FUNCTION_BLOCK "GCS7_GrpCtrlMain"	// FB 9
TITLE = Group Control UL
//
//COPYRIGHT:   (C) 1997 BY  BUHLER LTD
//                          CH-9240 UZWIL  SWITZERLAND
//
//PRODUCT:     GCS90
//
//TITLE:       FB 009 METHODS  OF  GROUPMANAGEMENT  with 320 groups
//                    Methoden der Gruppenverwaltung
//                    GCPROVB Revision =2
//-------------------------------------------------------------------------
//
//IDENT:        AUTOR:              DEPT:                           DATE:
//
//FB009.4.3     A.Egli              CT3                             23-Nov-2004
//              OutAutostartOkAll
//FB009.4.2     A.Egli              CT3                             14-Mar-2004
//              Reset Idling when group is externel used 
//FB009.4.1     A.Egli              CT3                             04-Mar-2004
//              Autostart: Filter with not ParNotRelForFault and 
//                                         ParNotRelForStarted
//FB009.4.0     A.Egli              CT3                             11-Nov-2003
//              OutAutoStartOkShared
//FB009.3.6     A.Egli              CT3                             14-Okt-2003
//              For available test use InExternal and not InLocked 
//FB009.3.5     A.Egli              CT3                             21-Aug-2003
//              Command OutAnyFault 
//FB009.3.4     A.Egli              CT3                             11-Aug-2003
//              Command CmdManualOffRel: 
//              Send command only to selected group, which OutShared=false
//FB009.3.3     A.Egli              CT3                             22-Jul-2003
//              Condition for All.OutStartWarning 
//FB009.3.2     A.Egli              CT3                             19-Mai-2003
//              OutStartwarning 
//FB009.3.1     A.Egli              CT3                             25-Mar-2003
//              OutPreStarted 
//FB009.3.0     A.Egli              CT3                             23-Sept-2002
//              New Relesae: 
//              OutLoaded;OutDPFault;OutHWStop;OutAutoStartOk; 
//              CmdContinue;InPreStart
//FB009.2.0     A.Egli              CT3                             13-Sept-2000
//              -320 group
//              -Any offset in section DB  
//              -Methode Code=0: Set Pointer 
//FB009.1.7     A.Egli              CT3                             13-Sept-2000
//              OutShared: Wrong pointer (DID with D replaced)
//FB009.1.6     A.Egli              CT3                             06-Jan-99
//              Warning if group with not rel. for fault is in state StFault
//FB009.1.5     A.Egli              CT3                             05-Jan-99
//              Warning if group with not rel. for fault is in state StFault
//FB009.1D      A.Egli              CT3                             20-Aug-99
//              OutFaultAll,FaultReset 
//FB009.1C      A.Egli              CT3                             18-Jul-99
//              OutWarning: Label wrong
//FB009.1B      A.Egli              CT3                             14-Okt-98
//              Reset InPreselected
//FB009.1A      A.Egli              AEE61                           13-Jun-96
//              1st Release
//
//-------------------------------------------------------------------------
//
//PURPOSE:            MANUAL : ....... .DOC
//                    CODE   : FB ...
//
//RESTRICTIONS: GCPROVB Revision >=2
//            
//-------------------------------------------------------------------------
//
//Calling convention:
//==================
//
//Actual open DB = Section DB
//
//Input parameter:
//===============
//CODE:
//  0 - Methode Set Pointer
//  1 - Methode InitPreselection
//  2 - Methode Selection
//  3 - Methode Deselection
//  4 - Methode UpdateCmdSt
//  5 - Methode UpdateEnable
//  6 - Methode UpdateOccupied
//
//Calling order for select of new groups:
//---------------------------------------
//1. Call Methode InitPreselection
//2. ASW: Prepare patter Sec.Gr.InPreselect 
//3. Call Methode Selection
//   ReturnValue: All.OutGrConflict
//4. Call ASW routine 'Select'
//
AUTHOR : EA
FAMILY : GCS7UL
NAME : GRVWMAIN
VERSION : 4.3
VAR_INPUT
  Code : INT ;	//0=Init,1=InitPreselect,2=Select,3=Deselect,4=UpdateCmdSt,5=UpdateEnable
END_VAR
VAR_IN_OUT
  Sec : UDT 20090;
END_VAR
VAR
  Spare : WORD ;
  All : STRUCT
   CmdClearIdling : BOOL ;	//Stop al groups of this section which are in idling
   OutAutoStartOkShared : BOOL ;
   InASWFlagAutostart : BOOL ;	//Free for ASW
   OutAutostartOkAll : BOOL ;	//Autostart of all selected groups ok
   Spare04 : BOOL ;
   Spare05 : BOOL ;
   OutPreStarted : BOOL ;
   OutPreStarting : BOOL ;	//Any group is pre-starting
   Spare10 : BOOL ;
   CmdContinue : BOOL ;	//(*new*)
   CmdManualOffRel : BOOL ;	//(*new*)
   CmdFaultReset : BOOL ;	//Command to fault reset
   CmdManualOff : BOOL ;	//Switch off maunual mode of all object
   OutStartwarning : BOOL ;	//Any selected group is in startwarning mode
   OutManualAny : BOOL ;	//Any object of this PLC is in manual mode
   InOutASWSelectionOK : BOOL ;	//Used by ASW
   OutSelectionValid : BOOL ;	//Any object is occupied for this section
   CmdNewSelection : BOOL ;	//An new object is occupied
   OutGrConflict : BOOL ;	//An object is not available
   OutGrIsLocked : BOOL ;	//An object is locked by ASW
   OutAutoStartOk : BOOL ;	//(*new*) All relevant Groups are in mode AutoStart
   OutManual : BOOL ;	//Any object of this section is in manual mode
   OutDPFault : BOOL ;	//(*new*)
   OutHWStop : BOOL ;	//(*new*)
   OutStoppedRel : BOOL ;
   OutStoppedAll : BOOL ;
   OutLoaded : BOOL ;	//(*new*)
   OutFaultIdling : BOOL ;
   OutFaultRel : BOOL ;
   OutFaultAll : BOOL ;
   OutIdling : BOOL ;
   OutWarning : BOOL ;
  END_STRUCT ;
  Feed : STRUCT
   InEnable : BOOL ;
   Spare01 : BOOL ;
   CmdNext : BOOL ;
   Spare03 : BOOL ;
   Spare04 : BOOL ;
   Spare05 : BOOL ;
   Spare06 : BOOL ;
   Spare07 : BOOL ;
   OutStoppedRel : BOOL ;
   OutStoppedAll : BOOL ;
   OutStartedRel : BOOL ;
   OutFaultIdling : BOOL ;
   OutFaultRel : BOOL ;
   OutFaultAll : BOOL ;
   OutIdling : BOOL ;
   OutSelected : BOOL ;
  END_STRUCT ;
  Mgr : STRUCT
   InEnable : BOOL ;
   Spare01 : BOOL ;
   CmdNext : BOOL ;
   Spare03 : BOOL ;
   Spare04 : BOOL ;
   Spare05 : BOOL ;
   Spare06 : BOOL ;
   Spare07 : BOOL ;
   OutStoppedRel : BOOL ;
   OutStoppedAll : BOOL ;
   OutStartedRel : BOOL ;
   OutFaultIdling : BOOL ;
   OutFaultRel : BOOL ;
   OutFaultAll : BOOL ;
   OutIdling : BOOL ;
   OutSelected : BOOL ;
  END_STRUCT ;
  Wgr : STRUCT
   InEnable : BOOL ;
   Spare01 : BOOL ;
   CmdNext : BOOL ;
   Spare03 : BOOL ;
   Spare04 : BOOL ;
   Spare05 : BOOL ;
   Spare06 : BOOL ;
   Spare07 : BOOL ;
   OutStoppedRel : BOOL ;
   OutStoppedAll : BOOL ;
   OutStartedRel : BOOL ;
   OutFaultIdling : BOOL ;
   OutFaultRel : BOOL ;
   OutFaultAll : BOOL ;
   OutIdling : BOOL ;
   OutSelected : BOOL ;
  END_STRUCT ;
  Ggr : STRUCT
   InEnable : BOOL ;
   Spare01 : BOOL ;
   CmdNext : BOOL ;
   Spare03 : BOOL ;
   Spare04 : BOOL ;
   Spare05 : BOOL ;
   Spare06 : BOOL ;
   Spare07 : BOOL ;
   OutStoppedRel : BOOL ;
   OutStoppedAll : BOOL ;
   OutStartedRel : BOOL ;
   OutFaultIdling : BOOL ;
   OutFaultRel : BOOL ;
   OutFaultAll : BOOL ;
   OutIdling : BOOL ;
   OutSelected : BOOL ;
  END_STRUCT ;
  InPreselect : ARRAY  [1 .. 320 ] OF BOOL ;
  OutSelected : ARRAY  [1 .. 320 ] OF BOOL ;
  OutIdling : ARRAY  [1 .. 320 ] OF BOOL ;
  ParNotRelForStarted : ARRAY  [1 .. 320 ] OF BOOL  := TRUE;
  ParNotRelForFault : ARRAY  [1 .. 320 ] OF BOOL  := TRUE;
  InManual : ARRAY  [1 .. 320 ] OF BOOL  := FALSE;
  InPreStart : ARRAY  [1 .. 320 ] OF //Input from section: These groups are pre-starting
  BOOL  := FALSE;
END_VAR
VAR_TEMP
  TmpInOut : STRUCT 	//Methode 4:Temporare copy of input an output of the actual type
   InEnable : BOOL ;
   Spare01 : BOOL ;
   CmdNext : BOOL ;
   Spare03 : BOOL ;
   Spare04 : BOOL ;
   InManual : BOOL ;
   Spare06 : BOOL ;
   Spare07 : BOOL ;
   OutStoppedRel : BOOL ;
   OutStoppedAll : BOOL ;
   OutStartedRel : BOOL ;
   OutFaultIdling : BOOL ;
   OutFaultRel : BOOL ;
   OutFaultAll : BOOL ;
   OutIdling : BOOL ;
   OutSelected : BOOL ;
  END_STRUCT ;
  tmpAddrInOut : DINT ;	//Methode 4: Address of TmpInOut
  VarSelGrActType : DWORD ;	//Methode 4: Temporare pattern
  VarSelGrActTypeId : DWORD ;	//Methode 4: Temporare pattern Selected +idling
  tmpValue : DINT ;
  tmpCntLoopGr : BYTE ;
  tmpCntLoopType : BYTE ;
  tmpAddrLoop : DWORD ;
  tmpAddrSecPreselect : DWORD ;
  tmpAddrSecSelected : DWORD ;
  tmpAddrSecIdling : DWORD ;
  tmpAddrSecManual : DWORD ;
  tmpAddrSecParRelStarted : DWORD ;
  tmpAddrSecParRelFault : DWORD ;
  tmpAddrDB9ParXxx : DWORD ;	//Pointer parameter of group of type xxxx
  tmpAddrDB9ParXxxLoop : DWORD ;
  tmpAddrSecInPreStart : DWORD ;
  tmpCODE : INT ;	//FUNC
  SecArray : DINT ;	//Pointer to Array DB9.Section
  SecDB : INT ;	//Actual section DB
  tmpOffsetDI : DINT ;	//Offset Instanz
  tmpCodeIs5 : BOOL ;	//Methode Update Enable
  tmpSecByteNr : DINT ;
  tmpStoreAR2 : DWORD ;
  tmpInstanzDB : INT ;
  tmpNotRelevant : DWORD ;
  tmpNotRelevantForFault : DWORD ;
END_VAR
BEGIN
NETWORK
TITLE = Init Part 1
      L     #Code;
      T     #tmpCODE;
      L     P##Sec;
      LAR1;
//--- Section DB of actual instanz ----------
      L     W [AR1,P#0.0];
      T     #SecDB;
//--- Set Pointer to instanz in section DB ----------
      L     D [AR1,P#2.0];
      SLD   8;
      SRD   11;
      T     #tmpSecByteNr;
//------------------------------
      L     #tmpCODE;
      L     5;	// do not init for methode "Update Enable"
      ==I;
      =     #tmpCodeIs5;
      JC    InEn;
//--- Call Section DB ----------
      OPN   DI [#SecDB];
      L     #tmpSecByteNr;
      SLD   3;
      L     P##Code;
      +D;
      L     P##All;	//) Section DB has only UDT20090
      SLD   8;	//) Correction AR2 (10 Byte)
      SRD   8;	//)
      -D;	//)
      LAR2;	//-->Instanz
InEn: TAR2  #tmpStoreAR2;
NETWORK
TITLE = Methode "Set Pointer"
//=======================================================================
      OPN   "GCS7_GrCtrlDB";
      L     #tmpCODE;
      L     0;
      <>I;
      JC    iEnd;
//==========================================================
//Check DB9.ParMaxGroupCnt    : must be between 1 and 10
      L     10;
      L     "GCS7_GrCtrlDB".ParMaxGroupCnt;
      <I;
      JC    Stop;
      L     1;
      <I;
      JC    Stop;
//=======================================================================
//Enter ByteNumber in DB9.Section[x].DBB [<--2.0
      L     "GCS7_GrCtrlDB".ParByteNoSecDB;	// ) ParByteArraySectionDB
      SLD   3;
      LAR1;
iSLo: L     W#16#FFFF;	// )=  Sektion-List
      L     DBW [AR1,P#0.0];	// )
      ==I;
      JC    iAdd;	//-->Add pointer, if pointer is not found
      L     DINO;	//-->Actual Section-DB
      ==I;
      JC    iSOt;	//-->Enter pointer
      +AR1  P#4.0;
      JU    iSLo;
//=======================================================================
//"Add DB-Pointer"
iAdd: L     #SecDB;	//Bit-Number Section Interface
      T     DBW [AR1,P#0.0];	//DB9.Section[n].DBB
      L     W#16#FFFF;
      T     DBW [AR1,P#4.0];	//DB9.Section[n+1].DBB
//=======================================================================
//"Set Pointer"
iSOt: L     #tmpSecByteNr;	//Bit-Number Section Interface
      T     DBW [AR1,P#2.0];	//DB9.Section[x].DBB
      BEU;
//=======================================================================
//!!!!Call Stop, if DB is not found or AR2 < P#DIX2.0   !!!!!!!
//Note: 1. Check DB9.Section[x].DBB    : must be >1
//      2. Check DB9.ParMaxGroupCnt    : must be between 1 and 10
Stop: CALL  "SIEMENS_STP";
//=======================================================================
iEnd: NOP   0;
NETWORK
TITLE = Code=1: Methode "InitPreselection"
      L     #tmpCODE;	// )
      L     1;	// )
      <>I;	// )
      JC    aEnd;	// )
//-----------------------------------
//Init InPreselect
//Init InPreStart
      LAR1  AR2;
      L     P##InPreselect;
      +AR1;
      L     "GCS7_GrCtrlDB".ParMaxGroupCnt;
F1LE: T     #tmpCntLoopGr;
// Reset enable bit of selected groups
      L     0;
      T     DID [AR1,P#0.0];	//  )-> InPreselect
      T     DID [AR1,P#240.0];	//  )-> InPreStart (P#262.0- P#22.0 =+240.0)
      +AR1  P#4.0;
      L     #tmpCntLoopGr;
      LOOP  F1LE;
      JU    BACK;
aEnd: NOP   0;
NETWORK
TITLE =  FUNC=2: meth. "selection"
      L     #tmpCODE;
      L     2;
      <>I;
      JC    F2En;
//--- Available test--------   
      R     #All.OutGrConflict;
      R     #All.OutGrIsLocked;
      R     #All.CmdNewSelection;
      R     #All.OutPreStarting;
      OPN   "GCS7_GrCtrlDB";
      LAR1  P#0.0;	// Pointer to DB9
//=======================================================================
// 1. Test New Selection: 
// ---------------------
// 1.0 Set OutPreStarting
// 1.1 Set idling 
// 1.2 Test available
// 1.3 Deleselect Conficted groups 
// 1.4 Deselect not used groups
//=======================================================================
//==Begin Loop Goups A                  ===
      L     "GCS7_GrCtrlDB".ParMaxGroupCnt;
F2L1: T     #tmpCntLoopGr;
//--Pointer section
      TAR1;
      TAR2;
      +D;
      T     #tmpOffsetDI;
      L     P##InPreselect;
      +D;
      T     #tmpAddrSecPreselect;
// 
      L     #tmpOffsetDI;
      L     P##OutSelected;
      +D;
      T     #tmpAddrSecSelected;
// 
      L     #tmpOffsetDI;
      L     P##OutIdling;
      +D;
      T     #tmpAddrSecIdling;
// 
      L     #tmpOffsetDI;
      L     P##InPreStart;
      +D;
      T     #tmpAddrSecInPreStart;
// 
// 1.0 Set OutPreStarting -----------
      L     DID [#tmpAddrSecInPreStart];	// Sec.InPreStart
      L     0;
      <>D;
      S     #All.OutPreStarting;
// 
// 1.1 Set idling -----------
      L     DID [#tmpAddrSecPreselect];	// Sec.InPreseleced
      INVD;
      L     DID [#tmpAddrSecSelected];	// Sec.OutSelected
      AD;	//-> not longer used groups
      L     DID [#tmpAddrSecIdling];	// Sec.OutIdling
      OD;
      T     DID [#tmpAddrSecIdling];	// Sec.OutIdling
// 1.2 Test available ----- 
      L     DID [#tmpAddrSecPreselect];
      L     DID [#tmpAddrSecSelected];
      <>D;
      S     #All.CmdNewSelection;
      INVD;
      AD;	// ==> new preseleted groups
      L     DBD [AR1,P#250.0];	// DB9.OutOccupied
      AD;	// ==> allready used groups
      L     DBD [AR1,P#170.0];	// DB9.ParShare
      INVD;
      AD;
      JN    F2C1;	//-->way conflict
      L     DID [#tmpAddrSecPreselect];
      L     DBD [AR1,P#690.0];	// DB9.InExternal  [3.5]
      AD;	// ==> allready used groups
      L     DBD [AR1,P#170.0];	// DB9.ParShare
      INVD;
      AD;
      JN    F2C1;	//-->way conflict
      L     DID [#tmpAddrSecPreselect];	//                          [3.6]
      L     DBD [AR1,P#650.0];	// DB9.InLocked             [3.6]
      AD;	// ==> allready used groups [3.6]
      L     DBD [AR1,P#170.0];	// DB9.ParShare             [3.6]
      INVD;	//                          [3.6]
      AD;	//                          [3.6]
      JN    F2C2;
      JU    F2Lx;
//----------------------------------
//Store groups with way conflict
F2C2: SET;
      S     #All.OutGrIsLocked;
      JU    F2Lx;
F2C1: SET;
      S     #All.OutGrConflict;
      S     #All.CmdNewSelection;
      T     DBD [AR1,P#970.0];	//  DB9.OutGrConflictObj 
// 
// 1.3 Deleselect Conficted groups 
      INVD;
      L     DID [#tmpAddrSecSelected];	// Sec.OutSelected
      AD;
      T     DID [#tmpAddrSecSelected];	// Sec.OutSelected
// Store DB
      L     DINO;
      T     "GCS7_GrCtrlDB".OutConflictSecDB;	//DB9.OutConflictSecDB
// 
//----------------------------------
// 1.4 Deselect not used groups
F2Lx: L     DID [#tmpAddrSecPreselect];	// Sec.InPreseleced
      L     DID [#tmpAddrSecSelected];	// Sec.OutSelected
      AD;
      T     DID [#tmpAddrSecSelected];	// Sec.OutSelected
//----------------------------------
      +AR1  P#4.0;	//->(next 32 groups)
      L     #tmpCntLoopGr;
      LOOP  F2L1;
//=End Loop Goups A                     === 
//=========================================
//=======================================================================
// 2. Copy Preselected   --> Selected  
//=======================================================================
//Select new groups
      A     #All.OutGrConflict;
      ON    #All.CmdNewSelection;
      JC    F2X2;
//--Begin Loop Groups B
      LAR1  AR2;
      L     "GCS7_GrCtrlDB".ParMaxGroupCnt;
F2L2: T     #tmpCntLoopGr;
//-Pointer
      TAR1;
      L     P##InPreselect;
      +D;
      T     #tmpAddrSecPreselect;
      TAR1;
      L     P##OutSelected;
      +D;
      T     #tmpAddrSecSelected;
//--Copy Preselected   --> Selected  
      L     DID [#tmpAddrSecPreselect];	// Sec.InPreseleced
      T     DID [#tmpAddrSecSelected];	// Sec.OutSelected
//--Next 32 groups 
      +AR1  P#4.0;
      L     #tmpCntLoopGr;
      LOOP  F2L2;
//--End Loop Groups B
//---------------------------------
F2X2: AN    #All.OutGrConflict;
      AN    #All.OutSelectionValid;
      S     #All.OutSelectionValid;
      JC    F5;	//--> Call Methode 6 "Update Occupied"
//=========================================
      A     #All.CmdNewSelection;
      JC    F5;	//--> Call Methode 6 "Update Occupied"
      JU    BACK;
F2En: NOP   0;
NETWORK
TITLE =  FUNC=3: meth. "Deselection all"
      L     #tmpCODE;
      L     3;
      <>I;
      JC    F3En;
      R     #All.OutGrConflict;
      R     #All.OutGrIsLocked;
      R     #All.CmdNewSelection;
//!!! Do only operate, if OutSelectionValid=true
      AN    #All.OutSelectionValid;
      JC    BACK;
      R     #All.OutSelectionValid;
//________________________________________
// -Copy Selected --> Idling  
// Begin Loop A
      LAR1  AR2;
      L     "GCS7_GrCtrlDB".ParMaxGroupCnt;
F3Lo: T     #tmpCntLoopGr;
//-Pointer
      TAR1;
      L     P##InPreselect;
      +D;
      T     #tmpAddrSecPreselect;
// 
      TAR1;
      L     P##OutSelected;
      +D;
      T     #tmpAddrSecSelected;
// 
      TAR1;
      L     P##OutIdling;
      +D;
      T     #tmpAddrSecIdling;
// 
      L     DID [#tmpAddrSecSelected];	// Sec.OutSelected
      L     DID [#tmpAddrSecIdling];	// Sec.OutIdling
      OD;
      T     DID [#tmpAddrSecIdling];	// Sec.OutIdling
      L     0;	//    
      T     DID [#tmpAddrSecPreselect];	// Sec.InPreseleced
      T     DID [#tmpAddrSecSelected];	// Sec.OutSelected
      +AR1  P#4.0;	//-> Next DD in section DB (next 32 groups) 
      L     #tmpCntLoopGr;
      LOOP  F3Lo;
// END Loop A
//   --Update DB9: Occupied -----
      JU    F5;	// Call Methode UpdateOcupied
F3En: NOP   0;
NETWORK
TITLE =  CODE=5: Methode "UpdateEnable", CODE=6"Update Occupied"
//Update DB9.OutEnable
//Update DB9.OutManual
//Update DB9.OutOccupied
//Update DB9.OutShared
//
//Is called aloso by methode 2: "Select" 
//Is called aloso by methode 3: "Deselect All" 
//
      L     #tmpCODE;
      L     5;	//Methode UpdateEnable
      ==I;
      JC    F5;
      L     #tmpCODE;
      L     6;	//Methode UpdateOccupied
      ==I;
      JC    F5;
      JU    F5En;
F5:   OPN   "GCS7_GrCtrlDB";
//=== Loop section ===========
      LAR1  P#DBX 0.0;	// Pointer to DB9
      L     "GCS7_GrCtrlDB".ParMaxGroupCnt;
F5L1: T     #tmpCntLoopGr;
// Reset enable bit of selected groups
      AN    #tmpCodeIs5;
      JC    F5J0;
      L     DBD [AR1,P#290.0];	// DB9.OutEnable 
      L     DBD [AR1,P#250.0];	// DB9.OutCccupied
      INVD;
      AD;
      T     DBD [AR1,P#290.0];	// DB9.OutEnable 
// Reset occupied bit
F5J0: L     0;	// 
      T     DBD [AR1,P#210.0];	// DB9.OutShared
      T     DBD [AR1,P#250.0];	// DB9.Occupied
//Next group
      +AR1  P#4.0;
      L     #tmpCntLoopGr;
      LOOP  F5L1;
//============================================
//Loop Section 
//============================================
      L     "GCS7_GrCtrlDB".ParByteNoSecDB;	// ) ParByteArraySectionDB
      SLD   3;
F5LS: T     #SecArray;
      L     W#16#FFFF;	// )=  Sektion-List
      L     DBW [#SecArray];	// DB9.Section[x].DBNr
      T     #tmpInstanzDB;	//-> Actual Section-DB
      ==I;
      JC    F5OT;	//-->Out
      L     0;
      ==I;
      JC    F5NS;	//--> Next section
      OPN   DI [#tmpInstanzDB];	//-->Pointer to instance in section
      LAR1  #SecArray;
      L     DBW [AR1,P#2.0];	//  DB9.Section[x].DBB
      SLD   3;
      L     P##Code;
      +D;
      L     P##All;	//) Section DB has only UDT20090
      SLD   8;	//) Correction AR2 (10 Byte)
      SRD   8;	//)
      -D;	//)
      LAR2;	//-->Pointer to instance in section
      LAR1  P#DBX 0.0;	// Pointer to DB9
//------------------------------------------
//Operate section x 
//------------------------------------------
      AN    #All.OutSelectionValid;	// )OutSelectionValid
      JC    F5NS;	// )
//-- Loop groups 
      L     "GCS7_GrCtrlDB".ParMaxGroupCnt;
F5LG: T     #tmpCntLoopGr;
// Pointer 
      TAR2;
      TAR1;
      +D;
      L     P##OutSelected;
      +D;
      T     #tmpAddrSecSelected;
// -- Occupied --
      L     DID [#tmpAddrSecSelected];	//  Sec.OutSelected
      L     DBD [AR1,P#250.0];	//  DB9.OutOccupied [1.7]
      AD;
      L     DBD [AR1,P#210.0];	//  DB9.OutShared
      OD;
      T     DBD [AR1,P#210.0];	//  DB9.OutShared
      L     DID [#tmpAddrSecSelected];	//  Sec.OutSelected
      L     DBD [AR1,P#250.0];	//  DB9.OutOccupied
      OD;
      T     DBD [AR1,P#250.0];	//->DB9.OutOccupied
//=== Enable ==============
      AN    #tmpCodeIs5;
      JC    F5XG;
// -- Enable Feed--
      AN    #Feed.InEnable;	// )Sec.Feed.InEnable
      JC    F5mg;	// )
      L     DID [#tmpAddrSecSelected];	// )Sec.OutSelected
      L     DBD [AR1,P#10.0];	// )DB9.ParFeed
      AD;	// )
      L     DBD [AR1,P#290.0];	// )DB9.OutEnable 
      OD;	// )(Set Enable)
      T     DBD [AR1,P#290.0];	// )DB9.OutEnable 
// -- Enable Mgr--
F5mg: AN    #Mgr.InEnable;	// )Sec.Mgr.InEnable
      JC    F5wg;	// )
      L     DID [#tmpAddrSecSelected];	// )Sec.OutSelected
      L     DBD [AR1,P#50.0];	// )DB9.ParMgr
      AD;	// )
      L     DBD [AR1,P#290.0];	// )DB9.OutEnable 
      OD;	// )(Set Enable)
      T     DBD [AR1,P#290.0];	// )DB9.OutEnable 
// -- Enable Wgr--
F5wg: AN    #Wgr.InEnable;	// )Sec.Wgr.InEnable
      JC    F5gg;	// )
      L     DID [#tmpAddrSecSelected];	// )Sec.OutSelected
      L     DBD [AR1,P#90.0];	// )DB9.ParWgr
      AD;	// )
      L     DBD [AR1,P#290.0];	// )DB9.OutEnable 
      OD;	// )(Set Enable)
      T     DBD [AR1,P#290.0];	// )DB9.OutEnable 
// -- Enable GGr--
F5gg: AN    #Ggr.InEnable;	// )Sec.Ggr.InEnable
      JC    F5XG;	// )
      L     DID [#tmpAddrSecSelected];	// )Sec.OutSelected
      L     DBD [AR1,P#130.0];	// )DB9.ParGgr
      AD;	// )
      L     DBD [AR1,P#290.0];	// )DB9.OutEnable 
      OD;	// )(Set Enable)
      T     DBD [AR1,P#290.0];	// )DB9.OutEnable 
F5XG: +AR1  P#4.0;
      L     #tmpCntLoopGr;
      LOOP  F5LG;
//=== End Loop groups ==
F5NS: L     #SecArray;
      L     P#4.0;
      +D;	// Pointer to next section
      JU    F5LS;
F5OT: OPN   DI [#SecDB];
      LAR2  #tmpStoreAR2;
F5En: NOP   0;
NETWORK
TITLE =  FUNC=4: meth. "UpdateCmdSt"
//- Update Sec.OutIdling[c]
//- Update Sec.xxx.OutIdling
//- Update Sec.xxx.OutSelected
//- Update State
//- Send Command to DB9
//Implementation: 
//--------------
//1.Part: Summery commands and state of all groups
//2.Part: State and commands of one type:
//  Because the function of Feed, Mgr, Wgr and GGr are nearly equal we use the 
//same code for all.
//  For this reason this segment is processed in a loop (5 times).
//  Loop 1: Feed
//  Loop 2: Mgr
//  Loop 3: Wgr
//  Loop 4: GGr
//
      L     #tmpCODE;
      L     4;
      ==I;
      JC    F4;
      L     #tmpCODE;
      L     2;
      ==I;
      JC    F4;
      JU    BACK;
F4:   R     #All.OutFaultIdling;	//-> Sec.All.OutIdlingFault
      R     #All.OutWarning;	//-> Sec.All.OutWarning
      R     #All.OutManual;	//-> Sec.All.OutManual
      R     #All.OutManualAny;	//-> Sec.All.OutManualAny
      R     #All.OutLoaded;	//[3.0]
      R     #All.OutDPFault;	//[3.0]
      R     #All.OutHWStop;	// [3.0]
      S     #All.OutAutoStartOk;	// [3.0]
      S     #All.OutAutoStartOkShared;	// [4.0]
      S     #All.OutAutostartOkAll;	// [4.3]
      S     #All.OutPreStarted;	//[3.0]
      R     #All.OutStartwarning;	// [3.0]
      R     "GCS7_GrCtrlDB".OutManualAny;	// [3.0]
      R     "GCS7_GrCtrlDB".OutFaultAny;	// [3.0]
//==Begin Loop Groups "summary" ===============================
      LAR1  P#0.0;	// Pointer to DB9.DX0.0
      L     "GCS7_GrCtrlDB".ParMaxGroupCnt;
F4L1: T     #tmpCntLoopGr;	//-->Loop counter groups
//---Pointer to section ---------------------------------------
      TAR1;
      TAR2;
      +D;
      T     #tmpOffsetDI;
      L     P##OutIdling;
      +D;
      T     #tmpAddrSecIdling;
      L     #tmpOffsetDI;
      L     P##OutSelected;
      +D;
      T     #tmpAddrSecSelected;
      L     #tmpOffsetDI;
      L     P##ParNotRelForFault;
      +D;
      T     #tmpAddrSecParRelFault;
      L     #tmpOffsetDI;
      L     P##ParNotRelForStarted;
      +D;
      T     #tmpAddrSecParRelStarted;	//[3.1]
      L     #tmpOffsetDI;
      L     P##InManual;
      +D;
      T     #tmpAddrSecManual;
      L     #tmpOffsetDI;
      L     P##InPreStart;
      +D;
      T     #tmpAddrSecInPreStart;
      L     DID [#tmpAddrSecInPreStart];
      L     DID [#tmpAddrSecParRelFault];	// )Sec.ParRelForFault
      OD;
      T     #tmpNotRelevantForFault;
//-- OutIdling --------------------------------------------
      L     DBD [AR1,P#250.0];	// ) DB9.OutOccupied
      L     DBD [AR1,P#690.0];	// ) DB9.InExternal             //[4.2]
      OD;
      L     DBD [AR1,P#450.0];	// ) DB9.InStopped
      OD;	// ) OR
      INVD;	// ) NOT
      L     DID [#tmpAddrSecIdling];	// ) Sec.OutIdling
      AD;	// )
      T     DID [#tmpAddrSecIdling];	// ) Sec.OutIdling
//--CmdContinue------------------------------------------- 
      AN    #All.CmdContinue;	// )Sec.CmdContinue [3.0]
      JC    F4CU;	// )                [3.0]
      L     DBD [AR1,P#730.0];	// )DB9.CmdContinue [3.0]
      L     DID [#tmpAddrSecSelected];	// )Sec.OutSelected [3.0]    
      OD;	// )                [3.0]
      T     DBD [AR1,P#730.0];	// )DB9.CmdContinue [3.0]
//--CmdManualOff------------------------------------------- 
F4CU: AN    #All.CmdManualOff;	// Sec.CmdManualOff
      JC    F4C2;	// 
      L     DBD [AR1,P#410.0];	// DB9.OutManualOff
      L     DID [#tmpAddrSecManual];	// Sec.InManual
      OD;	// 
      T     DBD [AR1,P#410.0];	// DB9.OutManualOff
//--CmdManualOff Relevant------------------------------------------- 
F4C2: AN    #All.CmdManualOffRel;	// Sec.CmdManualOff           //[3.4]
      JC    F4Fr;	//                            //[3.4]
      L     DBD [AR1,P#250.0];	// DB9.OutOccupied            //[3.4]  
      INVD;	// NOT                        //[3.4]  
      L     DID [#tmpAddrSecSelected];	// Sec.OutSelected            //[3.4]      
      OD;	//                            //[3.4]  
      L     DID [#tmpAddrSecManual];	// Sec.InManual               //[3.4]  
      AD;	//                            //[3.4]  
      T     #tmpValue;	// ==> not relevant group 
      L     DBD [AR1,P#690.0];	// DB9.InExternal             //[3.4]
      L     DBD [AR1,P#210.0];	// DB9.OutShared              //[3.4]
      OD;	//                            //[3.4]  
      INVD;	//                            //[3.4]  
      L     #tmpValue;	// not relevant group         //[3.4]  
      AD;	//                            //[3.4]  
      L     DBD [AR1,P#410.0];	// DB9.OutManualOff           //[3.4]  
      OD;	//                            //[3.4]  
      T     DBD [AR1,P#410.0];	// DB9.OutManualOff           //[3.4]  
//--CmdFaultReset------------------------------------------- 
F4Fr: AN    #All.CmdFaultReset;	// )Sec.CmdFaultReset
      JC    F4CI;
      L     DBD [AR1,P#250.0];	// ) DB9.OutOccupied    [1D]
      INVD;	// ) NOT                [1D]
      L     DID [#tmpAddrSecManual];	// )Sec.InManualGr      [1D]
      AD;	// )                    [1D]
      L     DID [#tmpAddrSecSelected];	// )Sec.OutSelected     
      OD;
      L     DBD [AR1,P#370.0];	// )DB9.CmdFaultReset
      OD;	// )
      T     DBD [AR1,P#370.0];	// )DB9.CmdFaultReset
//--- Clear idling ---------------------
F4CI: AN    #All.CmdClearIdling;	// )Sec.ClearIdling
      JC    F4MO;	// )
      L     DID [#tmpAddrSecIdling];	// )Sec.OutIdling
      INVD;	// )
      L     DBD [AR1,P#290.0];	// )DB9.OutEnable
      AD;	// )(Reset)
      T     DBD [AR1,P#290.0];	// )DB9.OutEnable
//--OutManual---    
F4MO: L     0;
      L     DBD [AR1,P#610.0];	// DB9.InManual
      <>D;
      S     #All.OutManualAny;	// 
      S     "GCS7_GrCtrlDB".OutManualAny;	// [3.0]
      SET;	// VKE must be 1 for all SPZ
      L     DID [#tmpAddrSecManual];	// Sec.InManualGr
      AD;	// 
      JZ    F4Wa;	// [1C]
      S     #All.OutManual;	//->
//--Warning---    
F4Wa: L     DID [#tmpAddrSecSelected];	// )Sec.OutSelected  [1C]
      L     DBD [AR1,P#570.0];	// )DB9.InWarning
      AD;	// )
      JZ    F4WO;	// )
      S     #All.OutWarning;	//->
//Waning if not rel for fault [Start rel 1.5]
F4WO: L     DID [#tmpAddrSecSelected];	// Sec.OutSelected  
      L     #tmpNotRelevantForFault;	// Sec.ParNotRelForFault /PreStart
      AD;	// )
      L     DBD [AR1,P#530.0];	// )DB9.InFault
      AD;	// )
      JZ    F4FI;	// )
      S     #All.OutWarning;	//-> [end rel. 1.5]
// --FaultAny    
F4FI: L     0;
      L     DBD [AR1,P#530.0];	// )DB9.InFault
      <>D;
      S     "GCS7_GrCtrlDB".OutFaultAny;	// [3.0]
// --FaultIdling    
      L     DID [#tmpAddrSecIdling];	// )Sec.OutIdling
      L     DBD [AR1,P#530.0];	// )DB9.InFault
      AD;	// )
      JZ    F4X1;	// )
      SET;
      S     #All.OutFaultIdling;	//-->Sec.All.OutFaultIdling
//--OutLoaded---    
F4X1: L     DID [#tmpAddrSecSelected];	// )Sec.OutSelected  [3.0]
      L     DBD [AR1,P#770.0];	// )DB9.OutLoaded    [3.0]
      AD;	// )                 [3.0]
      JZ    F4LD;	// )                 [3.0]
      SET;
      S     #All.OutLoaded;	//->                 [3.0]
//--OutDPFault---    
F4LD: L     DID [#tmpAddrSecSelected];	// )Sec.OutSelected  [3.0]
      L     DBD [AR1,P#810.0];	// )DB9.OutDPFault   [3.0]
      AD;	// )                 [3.0]
      JZ    F4DP;	// )                 [3.0]
      SET;
      S     #All.OutDPFault;	//->                 [3.0]
//--OutHWStop---    
F4DP: L     DID [#tmpAddrSecSelected];	// )Sec.OutSelected  [3.0]
      L     DBD [AR1,P#850.0];	// )DB9.OutHWStop    [3.0]
      AD;	// )                 [3.0]
      JZ    F4HS;	// )                 [3.0]
      SET;
      S     #All.OutHWStop;	//->                 [3.0]
//--OutAutoStartOk---    
F4HS: L     DID [#tmpAddrSecSelected];	// )Sec.OutSelected  [3.0]
      L     DID [#tmpAddrSecParRelStarted];	// ParNotRelForStarted [4.1]
      INVD;	//                    [4.1]
      AD;	//                    [4.1]
      L     #tmpNotRelevantForFault;	// Sec.ParRelForFault [4.1] 
      INVD;	//                    [4.1]
      AD;	//                    [4.1]
      L     DBD [AR1,P#890.0];	// )DB9.OutAutoStart [3.0]
      INVD;	// )                 [3.0]
      AD;	// )                 [3.0]
      JZ    F4A2;	// )                 [3.0]
      SET;
      R     #All.OutAutoStartOk;	//->                 [3.0]
//--OutAutoStartSharedOk---    
F4A2: L     DBD [AR1,P#690.0];	// DB9.InExternal    [4.0]
      L     DBD [AR1,P#210.0];	// DB9.OutShared     [4.0]
      OD;	//                   [4.0]
      L     DID [#tmpAddrSecParRelStarted];	// ParNotRelForStarted [4.1]
      OD;	//                    [4.1]
      L     #tmpNotRelevantForFault;	// Sec.ParRelForFault [4.1] 
      OD;	//                    [4.1] 
      L     DID [#tmpAddrSecSelected];	// Sec.OutSelected   [4.0]
      AD;	//                   [4.0]
      L     DBD [AR1,P#890.0];	// DB9.OutAutoStart  [4.0]
      INVD;	//                   [4.0]
      AD;	//                   [4.0]
      JZ    F4SW;	//                   [4.0]
      SET;	//                   [4.0]
      R     #All.OutAutoStartOkShared;	//->                 [4.0]
//--OutAutoStartOkAll---    
F4SW: L     DID [#tmpAddrSecSelected];	// Sec.OutSelected   [4.3]
      L     DBD [AR1,P#890.0];	// DB9.OutAutoStart  [4.3]
      INVD;	//                   [4.3]
      AD;	//                   [4.3]
      JZ    F4AA;	//                   [4.3]
      SET;	//                   [4.3]
      R     #All.OutAutostartOkAll;	//->                 [4.3]
//--OutStartwarning---    
F4AA: L     DID [#tmpAddrSecSelected];	// )Sec.OutSelected     [3.0]
      L     DBD [AR1,P#930.0];	// )DB9.OutStartwarning [3.0]
//[3.3]      INVD                              // )                    [3.0]
      AD;	// )                    [3.0]
      JZ    F4AS;	// )                    [3.0]
      SET;
      S     #All.OutStartwarning;	//->                 [3.0]
//------------------------------------------------------ 
//  --PreStarted                                      -----
F4AS: L     DBD [AR1,P#490.0];	// DB9.InStarted
      INVD;
      L     DID [#tmpAddrSecInPreStart];	// InPreStart
      AD;
      L     DID [#tmpAddrSecParRelStarted];	// ParNotRelForStarted
      INVD;
      AD;	// 
      JZ    F4SS;	// 
      SET;
      R     #All.OutPreStarted;
F4SS: +AR1  P#4.0;	//-> Next DD in DB9    (next 32 groups)
      L     #tmpCntLoopGr;
      LOOP  F4L1;
//==End Loop Groups "summary" =====================================
//=================================================================
// 4 Loops (FEED, MGR, WGR, GGR)
//=================================================================
// CntLoopTyp=0 : FEED
// CntLoopTyp=1 : MGR
// CntLoopTyp=2 : WGR
// CntLoopTyp=3 : GGR
// 
// Note:  'InOut' of the actual typeis copied to TmpInOut 
      L     P##TmpInOut;
      T     #tmpAddrInOut;
      L     0;
F4L2: T     #tmpCntLoopType;
      JL    H5xx;
      JU    HFe1;
      JU    HMg1;
      JU    HWg1;
      JU    HGg1;
H5xx: JU    HSav;	//-->Last type
//---- Copy Feed to Buffer ----------------
HFe1: L     P##Feed;
      TAR2;
      +D;
      T     #tmpAddrLoop;
      L     DIW [#tmpAddrLoop];	// Sec.Feed.InOut
      T     LW [#tmpAddrInOut];	// Buffer TmpInOut
      L     P#DBX 10.0;	// DB9.ParFeed
      T     #tmpAddrDB9ParXxx;
      JU    HCmd;	//--> Start 
//--- Store Buffer to Feed -----------------
HMg1: L     LW [#tmpAddrInOut];	//  Buffer TmpInOut
      T     DIW [#tmpAddrLoop];	//->Sec.Feed.InOut
//    Copy Mgr to Buffer
      L     P##Mgr;
      TAR2;
      +D;
      T     #tmpAddrLoop;
      L     DIW [#tmpAddrLoop];	//  Sec.Mgr.InOut
      T     LW [#tmpAddrInOut];	//  Buffer TmpInOut
      L     P#50.0;	//  DB9.ParMgr
      T     #tmpAddrDB9ParXxx;
      JU    HCmd;	//--> Start 
//--- Store Buffer to MGR -------------------
HWg1: L     LW [#tmpAddrInOut];	//CopyInOut
      T     DIW [#tmpAddrLoop];	//->Sec.Mgr.InOut
//--- Copy Wgr to Buffer
      L     P##Wgr;
      TAR2;
      +D;
      T     #tmpAddrLoop;
      L     DIW [#tmpAddrLoop];	//  Sec.Wgr.InOut
      T     LW [#tmpAddrInOut];	//  Buffer TmpInOut
      L     P#DBX 90.0;	//  DB9.ParWgr
      T     #tmpAddrDB9ParXxx;
      JU    HCmd;	//--> Start 
//--- Store Buffer to Wgr -------------------
HGg1: L     LW [#tmpAddrInOut];	//  Buffer TmpInOut
      T     DIW [#tmpAddrLoop];	//->Sec.Wgr.InOut
//--- Copy Ggr to Buffer --------------------
      L     P##Ggr;
      TAR2;
      +D;
      T     #tmpAddrLoop;
      L     DIW [#tmpAddrLoop];	//  Sec.Ggr.InOut
      T     LW [#tmpAddrInOut];	//  CopyInOut
      L     P#DBX 130.0;	//  DB9.ParGgr
      T     #tmpAddrDB9ParXxx;
      JU    HCmd;	//--> Start 
//--- Store Buffer to Ggr -------------------
HSav: L     LW [#tmpAddrInOut];	//CopyInOut
      T     DIW [#tmpAddrLoop];	//->Sec.Ggr.InOut
      JU    HOut;
//======================================================
//==Begin Loop groups                             ====== 
HCmd: LAR1  P#0.0;	// Pointer to DB9.DX0.0
      SET;
      S     #TmpInOut.OutStoppedRel;
      S     #TmpInOut.OutStoppedAll;
      S     #TmpInOut.OutStartedRel;
      R     #TmpInOut.OutFaultRel;
      R     #TmpInOut.OutFaultAll;
      R     #TmpInOut.OutIdling;
      R     #TmpInOut.OutSelected;
      L     "GCS7_GrCtrlDB".ParMaxGroupCnt;
HLo2: T     #tmpCntLoopGr;	// ) Loop Counter
//---------------------------
//Pointer to section 
      TAR1;
      TAR2;
      +D;
      T     #tmpOffsetDI;
      L     P##ParNotRelForStarted;
      +D;
      T     #tmpAddrSecParRelStarted;
      L     #tmpOffsetDI;
      L     P##ParNotRelForFault;
      +D;
      T     #tmpAddrSecParRelFault;
      L     #tmpOffsetDI;
      L     P##InPreStart;
      +D;
      T     #tmpAddrSecInPreStart;
      L     #tmpOffsetDI;
      L     P##OutIdling;
      +D;
      T     #tmpAddrSecIdling;
      L     #tmpOffsetDI;
      L     P##OutSelected;
      +D;
      T     #tmpAddrSecSelected;
      TAR1;
      L     #tmpAddrDB9ParXxx;
      +D;
      T     #tmpAddrDB9ParXxxLoop;
      L     DID [#tmpAddrSecInPreStart];
      L     DID [#tmpAddrSecParRelFault];	// )Sec.ParRelForFault
      OD;
      T     #tmpNotRelevantForFault;
//-- Selected 
      L     DID [#tmpAddrSecSelected];	// )Sec.OutSelected
      L     DID [#tmpAddrSecIdling];	// )Sec.OutIdling
      OD;
      L     DBD [#tmpAddrDB9ParXxxLoop];	// 
      AD;	// )
      T     #VarSelGrActTypeId;	//->selected+idling group of this type
      L     DBD [#tmpAddrDB9ParXxxLoop];	// 
      L     DID [#tmpAddrSecSelected];	// )Sec.OutSelected
      AD;	// )
      T     #VarSelGrActType;	//->selected group of this type
      JZ    HF1;
      S     #TmpInOut.OutSelected;	// )--> Sec.Feed.OutSelected
//------------------------------------------------------ 
//-- Selected / Idling                             -----
HF1:  L     DID [#tmpAddrSecIdling];	// ) Sec.OutIdling
      L     DBD [AR1,P#10.0];	// ) DB9.ParFeed
      AD;	// )
      JZ    HNx;
      S     #TmpInOut.OutIdling;	// )--> Sec.Feed.OutIdling
//------------------------------------------------------ 
//--CmdNext                                        ----- 
HNx:  AN    #TmpInOut.CmdNext;	// )Sec.xxx.CmdNext
      JC    HFa;
      L     #VarSelGrActType;	//->selected group of this type
      L     DBD [AR1,P#330.0];	// )DB9.CmdNext
      OD;	// )
      T     DBD [AR1,P#330.0];	// )DB9.CmdNext
//------------------------------------------------------ 
//  --FaultRel                                     -----
HFa:  L     #VarSelGrActType;	//->selected group of this type
      L     DBD [AR1,P#530.0];	// )DB9.InFault
      AD;	// )
      JZ    HSp;	// )
      S     #TmpInOut.OutFaultAll;	//-->Sec.xxx.FeedAny
      L     #tmpNotRelevantForFault;	// )Sec.ParRelForFault
      INVD;
      AD;	// )
      JZ    HSp;	// )
      S     #TmpInOut.OutFaultRel;	//-->Sec.xxx.FeedRel
//------------------------------------------------------ 
//  --Stopped                                      -----
HSp:  L     DBD [AR1,P#450.0];	// DB9.InStopped
      INVD;	// 
      L     #VarSelGrActTypeId;	// selected group of this type
      AD;	// 
      JZ    HSt;
      T     #tmpValue;	// ==> not stopped groups 
      R     #TmpInOut.OutStoppedAll;	//-->Sec.xxx.StoppedAll
      L     DBD [AR1,P#690.0];	// DB9.InExternal [2.0]
      L     DBD [AR1,P#210.0];	// DB9.OutShared
      OD;
      INVD;
      L     #tmpValue;	// <== not stopped groups 
      AD;
      JZ    HSt;
      R     #TmpInOut.OutStoppedRel;	//-->Sec.xxx.StoppedRel
//------------------------------------------------------ 
//  --Started                                      -----
HSt:  L     DID [#tmpAddrSecParRelStarted];	// ParRelForStarted
      L     DID [#tmpAddrSecInPreStart];	// InPreStart
      OD;
      T     #tmpNotRelevant;
      L     DBD [AR1,P#490.0];	// DB9.InStarted
      INVD;
      L     #VarSelGrActType;	// selected group of this type
      AD;
      L     #tmpNotRelevant;
      INVD;
      AD;	// 
      JZ    HStx;	// 
      R     #TmpInOut.OutStartedRel;	//-->Sec.xxx.Started
HStx: +AR1  P#4.0;	//-> Next DD in DB9    (next 32 groups)
      L     #tmpCntLoopGr;
      LOOP  HLo2;	//--> Next group commands (+4Byte)
//==End loop groups                       ==============
//======================================================
      SET;
      R     #TmpInOut.CmdNext;	// )Sec.xxx.CmdNext
      L     #tmpCntLoopType;
      +     1;
      JU    F4L2;
//========================================================================
// END Loops (FEED, MGR, WGR, GGR)
//=========================================================================
HOut: NOP   0;
      A     #Feed.OutStoppedRel;
      A     #Mgr.OutStoppedRel;
      A     #Wgr.OutStoppedRel;
      =     #All.OutStoppedRel;
      A     #Feed.OutStoppedAll;
      A     #Mgr.OutStoppedAll;
      A     #Wgr.OutStoppedAll;
      =     #All.OutStoppedAll;
      A     #Feed.OutFaultRel;
      O     #Mgr.OutFaultRel;
      O     #Wgr.OutFaultRel;
      O     #Ggr.OutFaultRel;
      =     #All.OutFaultRel;
      A     #Feed.OutFaultAll;
      O     #Mgr.OutFaultAll;
      O     #Wgr.OutFaultAll;
      O     #Ggr.OutFaultAll;
      =     #All.OutFaultAll;	// [1D]
      A     #Feed.OutIdling;
      O     #Mgr.OutIdling;
      O     #Wgr.OutIdling;
      O     #Ggr.OutIdling;
      =     #All.OutIdling;
      SET;
      R     #All.CmdFaultReset;
      R     #All.CmdManualOff;
      R     #All.CmdManualOffRel;	//[3.4]
      R     #All.CmdFaultReset;
      R     #All.CmdClearIdling;
      R     #All.CmdContinue;	// [3.0]
NETWORK
TITLE =  END
BACK: NOP   0;
END_FUNCTION_BLOCK

FUNCTION_BLOCK "GCS7_GrpCtrlSub"	// FB 10
TITLE = Group Help Function
//COPYRIGHT:    (C) 1996 BY  BUHLER LTD
//                          CH-9240 UZWIL  SWITZERLAND
//
//PRODUCT:      GCS7
//
//TITLE:        FB10  Group help function
//-------------------------------------------------------------------------
//
//IDENT:        AUTHOR:             DEPT:                       DATE:
//
//FB10.3.8       A. Egli             CT3                        28-Feb-2006
//              Reset CmdRestartIdling moved from Methode 2 to 1
//FB10.3.7       A. Egli             CT3                        20-Jan-2005
//              Methode 12: Store Changebit in Group
//FB10.3.6       A. Egli             CT3                        16-Nov-2004
//              Methode 12: Set Changebit
//FB10.3.5       A. Egli             CT3                        06-Okt-2004
//              12=Methode State Virtuell Group GCS90
//FB10.3.4       A. Egli             CT3                        17-Jun-2004
//              Reset Autostart as long OutHWStop or OutDPFault
//FB10.3.3       A. Egli             CT3                        12-Sep-2003
//              VarFlag1s , Reset delay for command CmdContinue of 1s
//FB10.3.2       A. Egli             CT3                        12-Sep-2003
//              Reset Autostart bits with CmdFaultReset when faulted
//FB10.3.1       A. Egli             CT3                        22-Jul-2003
//              Transition to StFault: Reset Autostart bits
//FB10.3.0       A. Egli             CT3                        09-Jan-2003
//              New release
//FB10.2.6       A. Egli             CT3                        23-Mar-2002
//              Examine: Call FC2  Methode 1 not 2
//FB10.2.5       A. Egli             CT3                        09-Feb-2001
//              GGR: Transition StStopping-->StStopped
//FB10.2E       A. Egli             CT3                         04-Aug-1999
//              GGR: Transition StStopped-->StStarted
//FB10.2D       S. Kalberer         CT3                         12-Jul-1999
//              CBIT in StStarting corrected
//FB10.2C       A. Egli             CT3                         19-Oct-1998
//              InSeqStop
//FB10.2B       S. Kalberer         CT3                         14-Oct-1998
//              R  M 13.6 (InHeavyStartup) deleted
//FB10.2A       A.Egli              CT3                         08-Jun-1998
//              StFault = StCode 32
//FB10.1B       A.Egli              AEE61                       29-Aug-1997
//              Code 2 for PC Direct Control
//FB10.1A       A.Egli              AEE61                        5-Jun-1996
//              1st Release
//
//-------------------------------------------------------------------------
//
//PURPOSE:      MANUAL : GRxxMAN.DOC             
//
//RESTRICTIONS: Before calling this FB, you have to select the requested
//              function code in the input variable 'tmpCode'.
//-------------------------------------------------------------------------
//
//Function Code:= tmpCode
//=============
//              1=Methode Control
//              2=Methode State
//             12=Methode State Virtuell Group GCS90   
AUTHOR : EA
FAMILY : GCS7LL
NAME : GrHlpFnc
VERSION : 3.8
VAR_INPUT
  FcCode : INT ;	//FunctionCode
END_VAR
VAR
  Spare2 : INT ;
  Spare4 : INT ;
  Spare6 : INT ;
  OutEmptyingTime : INT ;	//FB10: Actual Value Emptying Timer [s] (*NEW*)
  ChangeBit : STRUCT
   spare : BYTE ;
   CBit1 : BOOL ;
   CBit2 : BOOL ;
   CBit3 : BOOL ;
   CBit4 : BOOL ;
  END_STRUCT ;
  StCode : INT ;
  InEnableGr : BOOL ;	//Enable to run elemets of the group
  CmdContinue : BOOL ;	//Tick to restart after fault, Tick to start startwarning time (*NEW*)
  CmdRestartIdling : BOOL ;	//Restart idling time
  InReleaseEmptyingTime : BOOL ;	//ASW to FB10: Condiditon to run emptying time (*New*)
  InFeeding : BOOL ;	//ASW to FB10: Is used to set OutLoaded  (*NEW*)
  InOutAutostartMan : BOOL ;	//Autostart in manual mode: Whole machine starts
  InPreStart : BOOL ;	//ASW
  CmdManualOff : BOOL ;	//Switch off manual mode
  CmdOff : BOOL ;	//Tick to stop in manual mode
  CmdOn : BOOL ;	//Tick to start in manual mode
  CmdNext : BOOL ;	//Tick to start next element
  CmdFaultReset : BOOL ;	//Tick to rest fault
  InOccupied : BOOL ;	//Group is used in automatic mode
  InManual : BOOL ;	//Group is used in manual mode
  InLoadedSec : BOOL ;	//Loaded from section
  InSeqStop : BOOL ;	//Stop automatically after idling time
  ModePassive : BOOL ;	//Group is stopped AND not used
  ModeActive : BOOL ;	//Group is used
  ModeIdling : BOOL ;	//Group is not used, idling time running
  spare163 : BOOL ;
  spare164 : BOOL ;
  spare165 : BOOL ;
  spare166 : BOOL ;
  spare167 : BOOL ;
  StStopped : BOOL ;	//FB10:
  StStarting : BOOL ;	//FB10:
  StStarted : BOOL ;	//FB10:
  StStopping : BOOL ;	//FB10:
  StFault : BOOL ;	//FB10:
  OutLoaded : BOOL ;	//FB10: Is set by ASW, is reset by SSW  (*NEW*)
  OutWarning : BOOL ;	//ASW:
  OutFeeding : BOOL ;	//ASW:
  OutEnableEl : BOOL ;	//ASW: General condition to run element
  OutEnable1 : BOOL ;	//ASW:
  OutHWStop : BOOL ;	//FB10: Any used element has InHWStop (Copy of M15.0) (*NEW*)
  OutDPFault : BOOL ;	//FB10: Any used element has InDPFault(Copy of M15.1) (*NEW*)
  OutAutostart : BOOL ;	//FB10: Is set with command CmdStart , is reset with new fault (*NEW*)
  OutManual : BOOL ;	//FB10: Any object is in manual mode (Copy of M13.5)
  OutHornOn : BOOL ;	//FB10: Fault flag is set (Is set if M13.4 is true)
  OutEnablePrevGr : BOOL ;	//ASW:Enable to run previous group
  VarStopped : BOOL ;	//ASW to FB10: All relevant elements stopped
  VarStarted : BOOL ;	//ASW to FB10: All relevant elements started
  VarFault : BOOL ;	//ASW to FB10: A relevant element has fault
  VarStartwarning : BOOL ;	//ASW to FB10: Startwarning time is running
  VarFlag1s : BOOL ;
  OutEmptyingTimeDone : BOOL ;	//FB10 to ASW: (*New*)
  OutNewWay : BOOL ;	//FB10 to ASW:Read new pattern
  OutSeqStop : BOOL ;	//FB10 to ASW:Idling time end, Stop element
  OutIdlingTime : INT ;	//Actual idling time
  InCodePreselect : INT ;	//Free for user
  InLine : INT ;	//Line nr which use the line
  InCode : INT ;	//Target way or function
  OutCode : INT ;	//Actual way or function
  Par : STRUCT
   ParObjectNo : INT ;
   ParMgr : BOOL ;	//1=Machine group 0=Way group or general group
   ParWgr : BOOL ;	//1=Way group     0=Machine group or general group
   ParGgr : BOOL ;	//1=General group
   ParHornCode : INT ;	//Is used by horn module
   ParIdling : INT ;
   ParEmptyingTime : INT ;
   Para1_0 : BOOL ;
   Para1_1 : BOOL ;
   Para1_2 : BOOL ;
   Para1_3 : BOOL ;
   Para1_4 : BOOL ;
   Para1_5 : BOOL ;
   Para1_6 : BOOL ;
   Para1_7 : BOOL ;
   Para1_8 : BOOL ;
   Para1_9 : BOOL ;
   Para1_10 : BOOL ;
   Para1_11 : BOOL ;
   Para1_12 : BOOL ;
   Para1_13 : BOOL ;
   Para1_14 : BOOL ;
   Para1_15 : BOOL ;
   Para2 : INT ;
   Para3 : INT ;
   Para4 : INT ;
   Para5 : INT ;
  END_STRUCT ;
END_VAR
VAR_TEMP
  tmpAddr : DINT ;
END_VAR
BEGIN
NETWORK
TITLE = CODE 3: Emptying Time [3.0]
      L     #FcCode;
      L     3;
      <>I;
      JC    eEnd;
//------------------------------------
//Loaded
//------------------------------------
      A     #InFeeding;
      JCN   eJ0;
      S     #OutLoaded;
      R     #OutEmptyingTimeDone;
      L     0;
      T     #OutEmptyingTime;
      BEC;
//------------------------------------
//Check emptying time
//------------------------------------
eJ0:  L     #OutEmptyingTime;
      L     #Par.ParEmptyingTime;
      >=I;
      A     #InReleaseEmptyingTime;
      =     #OutEmptyingTimeDone;
      R     #OutLoaded;
      BEC;
//------------------------------------
//Run emptying time
//------------------------------------
      AN    #InReleaseEmptyingTime;
      ON    "GCS7_Gr_OutTick1s";
      BEC;
      L     #OutEmptyingTime;
      +     1;
      T     #OutEmptyingTime;
      BEU;
eEnd: NOP   0;
NETWORK
TITLE = CODE 4: Startwarning [3.0]
      L     #FcCode;
      L     4;
      <>I;
      JC    sEnd;
      BEU;
sEnd: NOP   0;
NETWORK
TITLE = Methode control: PC interface
      L     #FcCode;
      L     1;
      <>I;
      JC    aEnd;
//=== Test Object number =====================
      L     "SYS_DirectCtrlDB".PC.ObjectNo;	//Diag.ObjectNo
      L     #Par.ParObjectNo;	//Input ObjectNo
      <>I;
      JC    aEnd;
//=== Test OType      ========================
      L     3000;	//Input object type
      L     "SYS_DirectCtrlDB".PC.ObjectType;	//Diag.ObjectType
      <>I;
      JC    aEnd;
//=== Test Handshake =========================
      A     "SYS_DirectCtrlDB".PC.Hsk.FExamine;	// Handshake.FExamine
      JC    aExa;
      A     "SYS_DirectCtrlDB".PC.Hsk.FDefineCmd;	// Handshake.FDefineCmd
      JC    aCmd;
      A     "SYS_DirectCtrlDB".PC.Hsk.FDefinePara;	// Handshake.FDefinePara
      JC    pPar;
aIni: L     2;	// FcInit
      UC    "SYS_DirectCtrl";
      JU    aEnd;
// Write parameter 
pPar: LAR1  P#DBX 58.0;
      L     P#30.0;
      +AR1;
      L     DBW [AR1,P#6.0];
      T     #Par.ParIdling;
      L     DBW [AR1,P#8.0];
      T     #Par.ParEmptyingTime;
      L     DBW [AR1,P#10.0];
      T     DIW [AR2,P#40.0];
      L     DBW [AR1,P#12.0];
      T     #Par.Para2;
      L     DBW [AR1,P#14.0];
      T     #Par.Para3;
      L     DBW [AR1,P#16.0];
      T     #Par.Para4;
      L     DBW [AR1,P#18.0];
      T     #Par.Para5;
// Write new commands from PC to Interface of group 
aCmd: A     "SYS_DirectCtrlDB".PC.Cmd1[0];	//InEnableGr.On
      S     #InEnableGr;
      A     "SYS_DirectCtrlDB".PC.Cmd2[0];	//InEnableGr.Off
      R     #InEnableGr;
      A     "SYS_DirectCtrlDB".PC.Cmd1[8];	//CmdOff
      S     #CmdOff;
      A     "SYS_DirectCtrlDB".PC.Cmd1[9];	//CmdOn
      S     #CmdContinue;
      S     #CmdOn;
      A     "SYS_DirectCtrlDB".PC.Cmd1[10];	//CmdNext
      S     #CmdContinue;
      S     #CmdNext;
      A     "SYS_DirectCtrlDB".PC.Cmd1[11];	//CmdFaultReset
      S     #CmdFaultReset;
      A     "SYS_DirectCtrlDB".PC.Cmd1[12];	//InOccupied.On
      S     #InOccupied;
      A     "SYS_DirectCtrlDB".PC.Cmd2[12];	//InOccupied.Off
      R     #InOccupied;
      A     "SYS_DirectCtrlDB".PC.Cmd1[13];	//CmdManualOn
      S     #InManual;
      A     "SYS_DirectCtrlDB".PC.Cmd2[13];	//CmdManualOff
      S     #CmdManualOff;
      AN    "SYS_DirectCtrlDB".PC.Hsk.FDefinePara;	// Handshake.FDefineCmd
      JC    aIni;
      L     "SYS_DirectCtrlDB".PC.Value[23];	//Value[23]
      T     #Par.ParIdling;
      JU    aIni;
aExa: L     P##StCode;	// Address Dynamic datas
      T     "SYS_DirectCtrlDB".GC.InDynAddr;	// -->PCControl.GC.tmpDynAddr
      L     38;	// Length Dynamic datas
      T     "SYS_DirectCtrlDB".GC.InDynLen;	// -->PCControl.GC.tmpDynLen
      L     P##Par;	// Address Parameters
      T     "SYS_DirectCtrlDB".GC.InParaAddr;	// -->PCControl.GC.tmpParaAddr
      L     10;	// Lenth Parameter
      T     "SYS_DirectCtrlDB".GC.InParaLen;	// -->PCControl.GC.tmpParaLen
      L     1;	// Code FcExamine  [2.6]
      UC    "SYS_DirectCtrl";
aEnd: NOP   0;
NETWORK
TITLE = Methode control : Part Mode 
      L     #FcCode;
      L     1;
      <>I;
      JC    bEnd;
      R     "GCS7_Gr_InCBit1";	// Global.CBit1
      R     "GCS7_Gr_InCBit2";	// Global.CBit1
      R     "GCS7_Gr_InCBit3";	// Global.CBit1
      R     "GCS7_Gr_InCBit4";	// Global.CBit1
      R     "GCS7_Gr_InFault";	// Global.InFault
      R     "GCS7_Gr_InManual";	// Global.InManual
      R     "GCS7_Gr_InHWStop";	// Global.InHWStop"
      R     "GCS7_Gr_InDPFault";	// Global.InDPFault"
// Global.InHeavyStartup
      R     "GCS7_Gr_InFaultFlag";	// Global.InFaultFlag
      A     #CmdFaultReset;
      =     "GCS7_Gr_OutFaultReset";	// Global.OutFaultReset
//Autostart manual mode
      A     #InManual;
      A     #CmdOn;
      S     #InOutAutostartMan;
      AN    #InManual;
      O     #CmdOff;
      R     #InOutAutostartMan;
//CmdNext
      A     #InManual;
      R     #CmdNext;
      A     #InOutAutostartMan;
      O     #CmdOn;
      A     #InManual;
      S     #CmdNext;
      S     #InEnableGr;
      A     #CmdNext;
      =     "GCS7_Gr_OutNext";	// Global.OutNext
//InEnableGr
      AN    #InManual;
      JC    bJ1;
// Manual
      AN    #CmdOff;
      =     #InEnableGr;
//=====================
bJ1:  A     #CmdOff;
      R     #InEnableGr;
      A     #CmdManualOff;
      R     #InManual;
      =     "GCS7_Gr_OutManualOff";	// Global.OutManualOff
      L     #InLine;
      T     "GCS7_Gr_OutLine";
      L     #Par.ParHornCode;
      T     "Gr_ParHornCode";
      A     #ModeIdling;
      JC    MoId;	//  )=>ModeIdling 
      A     #ModeActive;
      JC    MoAc;	//  )=>ModeActive
//==Mode Passive ======================
      S     #ModePassive;
      S     #OutSeqStop;
      A     #InOccupied;
      O     #InManual;
      JC    TXAC;	//  )->Transition Active 
      JU    WAY;
//==Mode Idling  ======================
MoId: A     #InOccupied;
      O     #InManual;
      JC    TXAC;
      AN    #CmdRestartIdling;
      JC    ID1;
      L     #Par.ParIdling;
      T     #OutIdlingTime;
ID1:  AN    "GCS7_Gr_OutTick1s";
      L     #OutIdlingTime;
      JC    ID2;
      +     -1;
      T     #OutIdlingTime;
ID2:  L     0;
      <=I;
      =     #OutSeqStop;
      JCN   ID3;
      T     #OutIdlingTime;
ID3:  A     #StFault;
      O     #Par.ParWgr;
      A     #OutSeqStop;
      O     #StStopped;
      JCN   WAY;
//-- Transition to Passive----
      R     #ModeIdling;
      S     #ModePassive;
      L     0;	// )
      T     #OutIdlingTime;
      JU    CBit;
//=== ModeActive ================
MoAc: A     #InSeqStop;
      AN    #CmdRestartIdling;
      AN    #InManual;
      JC    ac1;
      L     #Par.ParIdling;
      T     #OutIdlingTime;
ac1:  AN    "GCS7_Gr_OutTick1s";
      O     #OutSeqStop;
      L     #OutIdlingTime;
      JC    ac2;
      +     -1;
      T     #OutIdlingTime;
ac2:  L     0;
      <=I;
      A     #InSeqStop;
      =     #OutSeqStop;
      JCN   ac3;
      T     #OutIdlingTime;
ac3:  A     #InOccupied;
      O     #InManual;
      JC    WAY;
//-- Transition to Idling -------
      S     #ModeIdling;
      R     #ModePassive;
      R     #ModeActive;
      L     #Par.ParIdling;
      T     #OutIdlingTime;
      JU    CBIT;	// 
//-- Transition to Active -------
TXAC: S     #ModeActive;
      R     #ModePassive;
      R     #ModeIdling;
      S     #OutNewWay;
      S     #OutAutostart;	//[3.0]
      R     #OutSeqStop;
      L     0;
      T     #OutIdlingTime;
CBit: SET;
      S     "GCS7_Gr_InCBit1";	// InChangeBit  
//Autostart
WAY:  A     #CmdContinue;	//[3.0]
      O     #ModePassive;
      S     #OutAutostart;	//[3.0]
//Reset OutAutostart                    //[3.2]
      A     #CmdFaultReset;	//[3.2]
      AN    #CmdContinue;	//[3.2]
      A     #VarFault;	//[3.2]
      R     #OutAutostart;	//[3.2]
      R     #InOutAutostartMan;	//[3.2]
      L     #OutCode;
      L     #InCode;
      T     #OutCode;
      <>I;
      S     #OutNewWay;
//Init
      SET;	//[3.8]
      R     #CmdRestartIdling;	//[3.8]
      BEU;
bEnd: NOP   0;
NETWORK
TITLE =  Methode State
//Interface to group:
//
//Inputs:
//- VarStopped
//- VarStarted
//- VarFault
//- VarEnableEl
//Outputs:
//-State
      L     #FcCode;
      L     2;
      <>I;
      JC    cEnd;	//3.5
      A     #StStarted;
      JC    ST2;
      A     #StStopping;
      JC    ST3;
      A     #StStarting;
      JC    ST1;
      A     #StFault;
      JC    ST4;
      A     #StStopped;
      JC    ST0;
      JU    NEWS;
// ===StStopped =========
ST0:  A     #VarFault;	// )
      JC    TX_4;	// )--> Transition to StFault
      A     #ModeActive;
      A     #OutEnableEl;
      A     #Par.ParWgr;
      O;
      AN    #VarStopped;
      A     #Par.ParMgr;
      O;	//[2E]
      A     #VarStarted;	//[2E]
      AN    #OutSeqStop;
      A     #OutEnableEl;
      AN    #Par.ParMgr;	//[2E]
      AN    #Par.ParWgr;	//[2E]
      JC    TX_1;	// )--> Transition to StStarting
      JU    Init;	// )
// == StStarting ==========================
ST1:  A     #VarFault;
      JC    TX_4;	// )--> transition to st_fault
      A     #VarStarted;
      JC    TX_2;	// )--> transition to st_started
      A(;	//  )
      A     #OutSeqStop;
      ON    #OutEnableEl;
      O;	// )
      A     #VarStopped;
      A     #Par.ParMgr;
      );	// )
      AN    #InManual;
      JC    TX_3;	//  )--> transition to st_stopping
      JU    Init;	// 2D: CBIT -> Init
// == StStarted ===========================
ST2:  A     #VarFault;
      JC    TX_4;	// )--> transition to st_fault
      A     #OutSeqStop;
      ON    #OutEnableEl;
      AN    #Par.ParMgr;
      ON    #VarStarted;
      JC    TX_3;	// )--> transition to st_stopping
      JU    Init;	// )
// == StStopping ============================
ST3:  A     #VarFault;
      JC    TX_4;	//  --> transition to st_fault
      AN    #Par.ParMgr;	//[2.5]
      AN    #Par.ParWgr;	//[2.5]
      O     #VarStopped;
      JC    TX_0;	// )--> transition to st_stopped
      AN    #OutSeqStop;
      A     #OutEnableEl;
      O     #InManual;
      JC    TX_1;	// )--> transition to st_starting
      JU    Init;
// == StFault   ============================
ST4:  A     #VarFault;
      JC    Init;
      JU    TX_3;	// --> transition to st_stopping
//=== Test Init State ===========
NEWS: A     #VarFault;
      JC    TX_4;	// --> transition to st_fault
      A     #VarStarted;
      JC    TX_2;	// --> transition to st_started
      A     #VarStopped;
      JC    TX_0;	// --> transition to st_stopped
      JU    TX_3;	// --> transition to st_stopping
//==== Transition ===============
TX_0: S     #StStopped;
      R     #StStopping;
      JU    CBIT;
// --> StStarting
TX_1: S     #StStarting;
      R     #StStopped;
      R     #StStopping;
      JU    CBIT;
// --> StStarted
TX_2: S     #StStarted;
      R     #StStarting;
      JU    CBIT;
// --> StStopping
TX_3: S     #StStopping;
      R     #StStarting;
      R     #StStarted;
      R     #StFault;
      JU    CBIT;
// -->StFault
TX_4: S     #StFault;
      R     #StStopped;
      R     #StStarting;
      R     #StStarted;
      R     #StStopping;
      R     #OutAutostart;	//[3.1]
      R     #InOutAutostartMan;	//[3.1]
CBIT: S     "GCS7_Gr_InCBit1";	// Global.InCBit1 
Init: NOP   0;
cEnd: NOP   0;
NETWORK
TITLE = State Virtuel Group GCS90S7 Part 1
      L     #FcCode;	//[3.5]
      L     12;	//[3.5]
      <>I;	//[3.5]
      JC    dEnd;	//[3.5] 
      R     "GCS7_Gr_InCBit1";	//[3.7] 
      R     "GCS7_Gr_InCBit2";	//[3.7] 
      R     "GCS7_Gr_InCBit3";	//[3.7] 
      R     "GCS7_Gr_InCBit4";	//[3.7] 
      L     #StCode;	//[3.5]
      L     32;	//[3.5]
      <>I;	//[3.5]
      A     #StFault;	//[3.5]
      O;	//[3.5]
      A     #CmdFaultReset;	//[3.5]
      AN    #CmdContinue;	//[3.5]
      A     #StFault;	//[3.5]
      R     #OutAutostart;	//[3.5]
      R     #InOutAutostartMan;	//[3.5]
      A     #CmdContinue;	//[3.5]
      ON    #InOccupied;	//[3.5]
      S     #OutAutostart;	//[3.5]
      SET;
      R     #CmdContinue;	//[3.5]
dEnd: NOP   0;
NETWORK
TITLE = State Code
// State                    StCode       Codetext
// ----------------------------------------------
// StFault                    32        fault
// StStopped                  1         stopped 
// StStarting                 2         starting
// StStarted                  3         started
// StStopping                 7         stopping
// StStoppedLocal            17         stopped 
//
      L     2;
      L     #FcCode;
      <>I;
      A(;	//3.5
      L     12;	//3.5
      <>I;	//3.5
      );	//3.5
      BEC;	//3.5
      A     #StStopped;
      A     #ModePassive;
      L     17;	// Code: stopped+Passive
      JC    STC;
      A     #StStopped;
      A     #VarStartwarning;
      L     11;	//Code: stopped.StartWarning
      JC    STC;
      A     #StStopped;
      L     1;	// Code: stopped
      JC    STC;
      A     #StStarting;
      L     2;	// Code: starting
      JC    STC;
      A     #StStarted;
      L     3;	// Code: started
      JC    STC;
      A     #StStopping;
      L     7;	// Code: stopping
      JC    STC;
      L     32;	// Code: fault
STC:  L     #StCode;	//[3.6]
      TAK;
      T     #StCode;	// Save state code
      <>I;
      S     "GCS7_Gr_InCBit1";	//[3.6] Global.InCBit1   
NETWORK
TITLE = Init
      L     #FcCode;	//[3.7]
      L     12;	//[3.7]
      ==I;	//[3.7]
      JC    M12C;
      L     #FcCode;	//[3.5]
      L     2;	//[3.5]
      <>I;	//[3.5]
      BEC;	//[3.5]
//Reset OutAutostart   [3.0]
      A     #CmdFaultReset;
      AN    #CmdContinue;	//[3.0]
      O     "GCS7_Gr_InFaultFlag";	//Global.InFaultFlag 
      A     #VarFault;
      O     "GCS7_Gr_InHWStop";	//Global.InHWStop" [3.4]
      O     "GCS7_Gr_InDPFault";	//Global.InDPFault" [3.4]
      R     #OutAutostart;	//[3.0]
      R     #InOutAutostartMan;
//Horn On
      A     "GCS7_Gr_InFaultFlag";	// Global.InFaultFlag 
      S     #OutHornOn;
//OutManual
      A     "GCS7_Gr_InManual";	// Global.InManual 
      O     #InManual;
      =     #OutManual;
//HWStop DPFault
      A     "GCS7_Gr_InHWStop";	// Global.InHWStop" [3.0]
      =     #OutHWStop;	//[3.0]
      A     "GCS7_Gr_InDPFault";	// Global.InDPFault" [3.0]
      =     #OutDPFault;	//[3.0]
//Reset command
      SET;
//[3.8]      R     #CmdRestartIdling
      R     #CmdOff;
      R     #CmdOn;
      R     #CmdNext;
      R     #CmdFaultReset;
      R     #CmdManualOff;
      R     #OutNewWay;
//Store CmdContinue for 1s
      A     "GCS7_Gr_OutTick1s";	//[3.3]
      A     #VarFlag1s;	//[3.3]
      R     #VarFlag1s;	//[3.3]
      R     #CmdContinue;	//[3.3]
      A     "GCS7_Gr_OutTick1s";	//[3.3]
      A     #CmdContinue;	//[3.3]
      S     #VarFlag1s;	//[3.3]
//Change bit
M12C: A     "GCS7_Gr_InCBit1";	// Global.InCBit1 
      S     #ChangeBit.CBit1;
      A     "GCS7_Gr_InCBit2";	// Global.InCBit2 
      S     #ChangeBit.CBit2;
      A     "GCS7_Gr_InCBit3";	// Global.InCBit3 
      S     #ChangeBit.CBit3;
      A     "GCS7_Gr_InCBit4";	// Global.InCBit4 
      S     #ChangeBit.CBit4;
END_FUNCTION_BLOCK

FUNCTION_BLOCK "GCS7_E_DigOutput"	// FB 11
TITLE = DigitalOutput
//  
//COPYRIGHT:    (C) 1996 BY  BUHLER LTD.
//                           CH-9240 UZWIL  SWITZERLAND
//
//PRODUCT:      GCS7
//
//TITLE:        Element Digital Output
//
//REVISION:     10
//
//-------------------------------------------------------------------------
//
//IDENT:        AUTHOR:             DEPT:                       DATE:
//
//FB11.4.1      A. Egli             CT3                         18-Jan-2006
//              Manual Mode: Reset Output when HWStop or DPFault 
//FB11.4.0      A. Egli             CT3                         17-Jun-2002
//              New Release with one block 
//FB11.3.4      A. Egli             CT3                         30-Aug-2001
//              Reset Output, if InLocal
//FB11.3.3      A. Egli             CT3                         29-Jun-2001
//              Reset Output, if InLocal
//FB11.3.2      A. Egli             CT3                         25-Mai-2000
//              StCode=8 == StStarted.Warning=8
//FB11.3.1      A. Egli             CT3                         18-Mai-2000
//              Condition for message warning
//FB11.3.0      A. Egli             CT3                         27-Apr-2000
//              OutWarning, ParDelayTime
//FB11.2D       A. Egli             CT3                          5-Jan-1999
//              OutpFaultReset
//FB11.2C       A. Egli             CT3                          2-Nov-1998
//              StStarting only by continuous valve
//FB11.2B       A. Egli             CT3                         17-Jul-1998
//              ParManual: Manual mode without interlocking
//              InSeqStop by ParPulsing
//FB11.2A       A. Egli             CT3                         04-Mai-1998
//              StFault = StCode 32
//              Global flag M12.2 (Gr.OutNext) removed
//FB11.1A       S. Kalberer         AEE61                       06-Aug-1997
//              1st Release in S7
//
//-------------------------------------------------------------------------
//
//PURPOSE:      MANUAL : see [DOxxMAN]
//
//RESTRICTIONS: S7
//              ACCU2: Pointer to dynamic datas of the element
//              ACCU1: Pointer to parameter datas of the element
//              CmdOff, CmdOn: always active
//
//-------------------------------------------------------------------------
//
//=======================================================
//Log Message: 
//------------------------------------------------------
// 0  stopped
// 2  started
// 9  fault cancelled
//10  fault device
//13  pre alarm fault (warning)
//
//=======================================================
//StCode:  State               
//------------------------------------------------------
//32  StFault                 
//41  Stopped.HWStop          StStopped + InHWStop 
//51  Stopped.DPFault         StStopped + DPFault
//61  Stopped.FaultDev        StStopped + InpFaultDev
// 1  StStopped               
// 2  StStarting              
// 3  StStarted               
// 5  StFalse                 
// 8  StStarted.Warning       
//
AUTHOR : EA
FAMILY : GCS7LL
NAME : DigOut
VERSION : 4.1
VAR
  StCode : INT ;	//Element state code
  InEnable : BOOL ;	//Enable to run the element (manual and automatic mode)
  spare0201 : BOOL ;
  InContinuous : BOOL ;	//Switch from pulsing signal to continuous signal
  spare0203 : BOOL ;
  spare0204 : BOOL ;
  spare0205 : BOOL ;
  InpRun : BOOL ;	//Only for filter
  InpFaultDev : BOOL ;	//Digital iniput: fault device
  CmdOff : BOOL ;	//Pulse to stop the element immediately (manual mode)
  CmdOn : BOOL ;	//Pulse to start the element (manual mode)
  CmdNext : BOOL ;	//Pulse to start the element in automatic mode (see global flags)
  CmdFaultReset : BOOL ;	//Command to reset fault
  InLocal : BOOL ;	//1= Local mode (no fault by start with service switch)
  InManual : BOOL ;	//1= Manual / 0= Automatic: Set and reset by PC
  InReport : BOOL ;	//Report of all state transitions
  InSeqStop : BOOL ;	//Stop automatically after idling time
  InHWStop : BOOL ;	//HW stop is detected, no fault
  InDPFault : BOOL ;	//DP-Fault is detected, no fault
  OutIdling : BOOL ;	//Idling is active
  OutWarning : BOOL ;	//Delay Time fault is running
  spare0404 : BOOL ;
  spare0405 : BOOL ;
  OutpFaultReset : BOOL ;	//Reset Alarm
  OutpRun : BOOL ;	//Digital output to run element
  StStopped : BOOL ;	//Element is stopped
  StStarting : BOOL ;	//Element is starting
  StStarted : BOOL ;	//Element is started
  spare0503 : BOOL ;
  StFault : BOOL ;	//Element has a fault
  StFalse : BOOL ;	//Element is in local mode and has a fault
  spare0506 : BOOL ;
  OutPausing : BOOL ;	//Pausing time is on (pulsing signal)
  OutAlarmNrLog : INT ;	//Last textnumber send to log
  Par : STRUCT
   ParObjectNo : INT ;	//Is used for communication with PC, e.g. for message
   ParMsgType : INT ;	//Is used for message (translation of state)
   ParHornCode : INT ;	//Is used by horn module
   ParLogOff : BOOL ;	//Report is Off
   ParManual : BOOL ;	//Manual mode without interlocking
   ParContinuous : BOOL ;	//Type with continuous signal
   ParPulse : BOOL ;	//Type with pulse signal
   ParPulsing : BOOL ;	//Type with pulsing signal
   ParFilter : BOOL ;	//Type is Filter
   ParOnTime : INT ;	//Starting time or length of pulse 'On'
   ParOffTime : INT ;	//Pausing time between to pulses
   ParIdlingTime : INT ;	//Requested idling time to stop motor in automatic mode
   ParDelayTime : INT ;	//Requested fault delay time
   OutTime : INT ;	//Actual value of timer
   OutDelayTime : INT ;	//Actual fault delay time
   spare26 : INT ;
   spare28 : INT ;
   InOutManPulseLen : INT ;	//Pulse length to start a the element
  END_STRUCT ;
END_VAR
VAR_TEMP
  tmpLOGvalue : WORD ;	//LOG value
  tmpLenDyn : DINT ;
  tmpReport : BOOL ;	//Global LOG all
  tmpEnable : BOOL ;	//Global LOG all
  tmpFault : BOOL ;
  tmpWarning : BOOL ;
  tmpLocal : BOOL ;
  tmpLocalFault : BOOL ;
END_VAR
BEGIN
NETWORK
TITLE =  Start Global
      L     34;
      T     #tmpLenDyn;	//--> Len dynamic data in byte
NETWORK
TITLE = PC Control
//=== Test Object number =====================
      L     "SYS_DirectCtrlDB".PC.ObjectNo;	//PCControl.ObjectNo
      L     #Par.ParObjectNo;	//Input ObjectNo
      <>I;
      JC    Ctrl;
//=== Test OType      ========================
      L     1011;	//Input object type
      L     "SYS_DirectCtrlDB".PC.ObjectType;	//PCControl.ObjectType
      <>I;
      JC    Ctrl;
//=== Test Handshake =========================
      A     "SYS_DirectCtrlDB".PC.Hsk.FExamine;	// Handshake.FExamine
      JC    pExa;
      A     "SYS_DirectCtrlDB".PC.Hsk.FDefineCmd;	// Handshake.FDefineCmd
      JC    pCmd;
      A     "SYS_DirectCtrlDB".PC.Hsk.FDefinePara;	// Handshake.FDefinePara
      JC    pPar;
pIni: L     2;	// FcInit
      UC    "SYS_DirectCtrl";
      JU    Ctrl;
// Write parameter 
pPar: LAR1  P#DBX 58.0;
      L     P##Par;
      L     DW#16#FFFFF;
      AD;
      +AR1;
      L     DBW [AR1,P#8.0];
      T     #Par.ParOnTime;
      L     DBW [AR1,P#10.0];
      T     #Par.ParOffTime;
      L     DBW [AR1,P#12.0];
      T     #Par.ParIdlingTime;
      L     DBW [AR1,P#14.0];
      T     #Par.ParDelayTime;
/// Write command 
pCmd: A     "SYS_DirectCtrlDB".PC.Cmd1[8];	// CmdOff
      S     #CmdOff;
      A     "SYS_DirectCtrlDB".PC.Cmd1[9];	// CmdOn
      S     #CmdOn;
      A     "SYS_DirectCtrlDB".PC.Cmd1[10];	// CmdNext
      S     #CmdNext;
      A     "SYS_DirectCtrlDB".PC.Cmd1[11];	// CmdFaultReset
      S     #CmdFaultReset;
      A     "SYS_DirectCtrlDB".PC.Cmd1[13];	// CmdManualOn
      S     #InManual;
      A     "SYS_DirectCtrlDB".PC.Cmd1[14];	// CmdReportOn
      S     #InReport;
      A     "SYS_DirectCtrlDB".PC.Cmd2[13];	// CmdManualOff
      R     #InManual;
      A     "SYS_DirectCtrlDB".PC.Cmd2[14];	// CmdReportOff
      R     #InReport;
      AN    "SYS_DirectCtrlDB".PC.Cmd1[1];	// CmdOnTik
      O     "GCS7_Gr_OutManualOff";	//Global.OutManualOff
      JC    pIni;
      L     "SYS_DirectCtrlDB".PC.Cmd3;	// "SYS_PCControl".PC.Cmd3
      T     #Par.InOutManPulseLen;
      JU    pIni;
pExa: TAR2;	// Address Dynamic datas
      T     "SYS_DirectCtrlDB".GC.InDynAddr;	// -->PCControl.GC.InDynAddr
      L     #tmpLenDyn;	// Length Dynamic datas
      T     "SYS_DirectCtrlDB".GC.InDynLen;	// -->PCControl.GC.InDynLen
      L     0;
      T     "SYS_DirectCtrlDB".GC.InParaAddr;	// -->PCControl.GC.InParaAddr
      T     "SYS_DirectCtrlDB".GC.InParaLen;	// -->PCControl.GC.InParaLen
      L     1;	// Code FcExamine
      UC    "SYS_DirectCtrl";
      L     10;	//Revision
      T     "SYS_DirectCtrlDB".GC.Revision;
NETWORK
TITLE =  All State Init
//===Global Group Orders===
Ctrl: A     "GCS7_Gr_OutManualOn";	//Global.OutManualOn
      S     #InManual;
      A     "GCS7_Gr_OutManualOff";	//Global.OutManualOff
      R     #InManual;
      A     #InManual;
      S     "GCS7_Gr_InManual";	//Global.InManualMode
      A     #Par.ParFilter;
      S     #Par.ParContinuous;
//tmpLocal
      A     #InLocal;
      AN    #InManual;
      =     #tmpLocalFault;	//[4.0]
      A     #tmpLocalFault;	//[4.0]
      O     #InHWStop;	//[4.0]
      O     #InDPFault;	//[4.0]
      =     #tmpLocal;
//---FaultReset Part 1---
      A     "GCS7_Gr_OutFaultReset";	// Gr.OutFaultReset
      S     #CmdFaultReset;
//---Report is on---
      O     "GCS7_Gr_OutReportAll";	//---Global OutReportAll
      O     #InReport;
      =     #tmpReport;
//--tmpEnable
      AN    #InManual;
      ON    #Par.ParManual;
      A     #InEnable;
      AN    #tmpLocal;	//3.4
      O;
      A     #InManual;
      A     #Par.ParManual;
      AN    #tmpLocal;	//[4.1]
      =     #tmpEnable;
//---Warning -----
//Warning time
      AN    #InpRun;
//        U  #InpFaultDev;    
      JC    glJ1;
      L     #Par.ParDelayTime;
      T     #Par.OutDelayTime;
      JU    glJ2;
glJ1: L     0;
      L     #Par.OutDelayTime;	// Set Timer
      >=I;
      ON    "GCS7_Gr_OutTick1min";	// Tick1Min
      ON    #OutpRun;
      JC    glJ2;
      +     -1;
      T     #Par.OutDelayTime;
glJ2: L     0;
      >I;
      O(;
      L     #Par.ParDelayTime;
      ==I;
      );
      A     #OutpRun;
      AN    #InpRun;
      AN    #StStopped;
      AN    #StStarting;
      AN    #StFault;
      A     #Par.ParFilter;
      FP    #OutWarning;
      =     #tmpWarning;
      AN    #tmpWarning;	//[3.1]
      O     #StFault;
      JC    glJ3;
      S     "GCS7_Gr_InFaultFlag";	// Gr.InFaultFlag
      CALL  "SYS_Horn_Code" (
           FcCode                   := 1,
           ParObjectType            := 1011,
           ParObjectNo              := #Par.ParObjectNo,
           ParHornCode              := #Par.ParHornCode);
//--- Message Warning ----------------------- 
      A     #Par.ParLogOff;	//---Set LOG Message
      JC    glJ3;
      L     B#(1, 13);	// MessageClass Warning
      T     #tmpLOGvalue;
      CALL  "GCS7_LogConvert" (
           ObjectNo                 := #Par.ParObjectNo,
           MsgType                  := #Par.ParMsgType,
           ClassMsgTxt              := #tmpLOGvalue,
           OType                    := 1011);	// LOG Message Converter / Entry / Contains Class and TextNo
//--Fault
glJ3: L     #Par.OutDelayTime;
      L     0;
      <=I;
      A     #OutpRun;
      AN    #InpRun;
      AN    #StStopped;
      AN    #StStarting;
      A     #Par.ParFilter;
      AN    #OutWarning;
      O;
      A     #InpFaultDev;
      AN    #tmpLocal;
      =     #tmpFault;
NETWORK
TITLE = Start as Pulse
      AN    #tmpEnable;
      ON    #InManual;
      O     #CmdOff;
      JC    STP1;
      L     0;
      L     #Par.InOutManPulseLen;
      >=I;
      JC    STP2;
      S     #CmdOn;
      AN    "GCS7_Gr_OutTick200ms";	// Decrement all 200ms
      JC    STP2;
      +     -2;
      T     #Par.InOutManPulseLen;
      L     0;
      >I;
      JC    STP2;
      S     #CmdOff;
STP1: L     0;
      T     #Par.InOutManPulseLen;
STP2: NOP   0;
NETWORK
TITLE = States
      A     #StStopped;	//===State machine===
      JC    S0;
      A     #StStarted;
      JC    S2;
      A     #StStarting;
      JC    S1;
      A     #StFault;
      JC    S4;
      A     #StFalse;
      JC    S5;
      S     #StStopped;	//Initialise: goto StStopped
      JU    S0;
NETWORK
TITLE = StStopped
//== Any Transition to StStarted
xxS0: SET;
      S     #StStopped;
      L     0;	// Reset actual timer value
      T     #Par.OutTime;
      AN    #tmpReport;	// ReportAll?
      JC    SAVE;
      L     B#(4, 0);	// MessageClass Info Stopped
      JU    LOG;
//==Logic ==== 
S0:   R     #OutIdling;
      A     #tmpFault;	//---Condition for StFault
      JC    S0J9;
      O     #CmdOff;	//---Condition for StStopped
      ON    #tmpEnable;
      JC    SAVE;
      AN    #InSeqStop;
      ON    #Par.ParContinuous;
      A     #CmdNext;	// Condition for StStarting
      AN    #InManual;
      O     #CmdOn;
      JC    S0J2;
      JU    SAVE;
S0J2: R     #StStopped;
      L     #Par.ParOnTime;	// Set actual vaule of timer
      T     #Par.OutTime;
      A     #Par.ParContinuous;
      S     #StStarting;	//---Transition -> StStarting
      JC    SAVE;
      JU    xxS2;	//---Transition -> StStarted
S0J9: R     #StStopped;	//---Transition -> StFault
      JU    xS45;
NETWORK
TITLE = StStarting
//StStarting: Only type continuous
S1:   A     #tmpFault;	//---Condition for StFault
      JC    S1J9;
      A     #InSeqStop;	//---Condition for StStopped
      AN    #InManual;
      ON    #tmpEnable;
      O     #CmdOff;
      JC    S1J3;
      AN    "GCS7_Gr_OutTick200ms";	//---Condition for StStarting
      L     #Par.OutTime;	// Set Timer
      JC    S1J1;
      +     -2;
      T     #Par.OutTime;
S1J1: L     0;
      >I;	// Starting time over
      JC    SAVE;
      R     #StStarting;	//---Transition -> StStarted
      JU    xxS2;
S1J3: R     #StStarting;	//---Transition -> StStopped
      JU    xxS0;
S1J9: R     #StStarting;	//---Transition -> StFault
      JU    xS45;
NETWORK
TITLE = StStarted
//== Any Transition to StStarted
xxS2: SET;
      S     #StStarted;
      AN    #tmpReport;	// ReportAll?
      JC    SAVE;
      L     B#(4, 2);	// MessageClass Info Started
      JU    LOG;
//==Logic ==== 
S2:   A     #tmpFault;	//---Condition for StFault
      JC    S2J9;
      AN    #tmpEnable;	//---Condition for StStopped
      O     #CmdOff;
      JC    S2J4;
      AN    #Par.ParPulse;	//---Type Pulse
      JC    S2J2;
      AN    "GCS7_Gr_OutTick200ms";	// Condition for StStarted
      L     #Par.OutTime;	// Set Timer
      JC    S2J1;
      +     -2;
      T     #Par.OutTime;
S2J1: L     0;	// Condition for StStopped
      <=I;
      JC    S2J4;
      JU    SAVE;	// stay in StStarted
S2J2: AN    #Par.ParPulsing;	//---Type Pulsing
      JC    S2J3;
      A     #InContinuous;	// pulsing -> continuous
      AN    #InManual;
      R     #OutPausing;
      JC    IDL1;
      AN    "GCS7_Gr_OutTick200ms";	// Condition for StStarted
      L     #Par.OutTime;	// Set Timer
      JC    OSC1;
      +     -2;
      T     #Par.OutTime;
OSC1: A     #OutPausing;	//---Condition for toggling
      JC    OSC2;
      L     0;	//---OnTime is active
      >I;
      JC    IDL1;
      S     #OutPausing;
      L     #Par.ParOffTime;	// Set actual vaule of timer
      T     #Par.OutTime;
      JU    IDL1;
OSC2: L     0;	//---OffTime is active
      >I;
      JC    IDL1;
      R     #OutPausing;
      L     #Par.ParOnTime;	// Set actual vaule of timer
      T     #Par.OutTime;
      JU    SAVE;
S2J3: O     #InSeqStop;	//---Type Continuous: Idling time 
      ON    #OutIdling;	// Condition to reset Idling-Time
      JC    IDL1;
      R     #OutIdling;
      L     0;
      T     #Par.OutTime;
      JU    SAVE;
IDL1: ON    #InSeqStop;	// Idling time active ?
      O     #InManual;
      JC    SAVE;
      A     #OutIdling;
      JC    IDL2;
      S     #OutIdling;	// Preset Idling Time
      L     #Par.ParIdlingTime;
      T     #Par.OutTime;
IDL2: AN    "GCS7_Gr_OutTick200ms";	// Set Idling Time
      L     #Par.OutTime;
      JC    IDL3;
      +     -2;
      T     #Par.OutTime;
IDL3: L     0;
      >I;	// Idling time over
      JC    SAVE;
S2J4: R     #StStarted;	//---Transition -> StStopped
      R     #OutPausing;
      JU    xxS0;
S2J9: R     #StStarted;	//---Transition -> StFault
      R     #OutPausing;
      JU    xS45;
NETWORK
TITLE =  StFault
// Any transiton to StFault/StFalse
xS45: L     0;	// Reset actual timer value
      T     #Par.OutTime;
      A     #tmpLocalFault;
      S     #StFalse;
      R     #StFault;
      JC    SAVE;
      S     #StFault;
      R     #StFalse;
      S     "GCS7_Gr_InFaultFlag";	// Gr.InFaultFlag
      CALL  "SYS_Horn_Code" (
           FcCode                   := 1,
           ParObjectType            := 1011,
           ParObjectNo              := #Par.ParObjectNo,
           ParHornCode              := #Par.ParHornCode);
S4S4: L     B#(1, 10);	// MessageClass Error fault
      JU    LOG;
//===logic StFault
//---Condition for StFalse
S4:   A     #tmpLocalFault;
      JC    xS45;
//-Wait for fault reset
      AN    "GCS7_Gr_OutTick500ms";	// Gr.OutTick500ms
      ON    #OutpFaultReset;
      JC    SAVE;
      R     #OutpFaultReset;
//---Condition for StFault with LOG
      A     #InpFaultDev;
      JC    S4S4;
//---Transition -> StStopped
      R     #StFault;
      S     #StStopped;
      L     B#(3, 9);	// MessageClass Operate fault cancelled
      JU    LOG;
NETWORK
TITLE =  StFalse
//Condition for StStopped
S5:   AN    #tmpFault;
      R     #StFalse;
      JC    xxS0;
//Condition for StFault
      AN    #tmpLocal;
      JC    xS45;
      JU    SAVE;
NETWORK
TITLE = LOG Message
LOG:  A     #Par.ParLogOff;	//---Set LOG Message
      JC    SAVE;
      T     #tmpLOGvalue;
      L     W#16#FF;
      AW;
      T     #OutAlarmNrLog;
      CALL  "GCS7_LogConvert" (
           ObjectNo                 := #Par.ParObjectNo,
           MsgType                  := #Par.ParMsgType,
           ClassMsgTxt              := #tmpLOGvalue,
           OType                    := 1011);	// LOG Message Converter / Entry / Contains Class and TextNo
NETWORK
TITLE = Global End
SAVE: NOP   0;
//===Set Output fault reset
      A     "GCS7_Gr_OutTick500ms";	// Gr.OutTick500ms
      AN    #StFault;
      R     #OutpFaultReset;
//===OutpFaultReset
      A     "GCS7_Gr_OutTick500ms";	// Gr.OutTick500ms
      A     #CmdFaultReset;
      S     #OutpFaultReset;
      R     #CmdFaultReset;
//OutpRun
//---Condition for setting output
      A     #CmdNext;	//[3.4]
      AN    #InManual;	//[3.4]
      O     #CmdOn;	//[3.4]
      O     #OutpRun;	//[3.4]
      A     #Par.ParFilter;
      A     #StFault;
      O     #StStarting;
      O     #StStarted;
      A     #tmpEnable;
      AN    #CmdOff;	//[3.4]
      AN    #OutPausing;
      =     #OutpRun;
//---Clear all commands
      CLR;
      =     #CmdOn;
      =     #CmdOff;
      =     #CmdNext;
//--Output for group 
      A     #InDPFault;
      AN    #tmpLocalFault;
      S     "GCS7_Gr_InDPFault";
      A     #InHWStop;
      AN    #tmpLocalFault;
      S     "GCS7_Gr_InHWStop";
NETWORK
TITLE = State Code
//--Stopped, Substate ---
      AN    #StStopped;
      JC    STC1;
      L     41;	//Code: StStopped.HWStop
      A     #InHWStop;
      JC    STC9;
      L     51;	//Code: StStopped.DPFault
      A     #InDPFault;
      JC    STC9;
      A     #InpFaultDev;	// [3.0]
      L     61;	// [3.0]
      JC    STC9;	// [3.0]
      L     1;	// Code: StStopped
      JU    STC9;
//--------------------
STC1: AN    #StStarted;
      JC    STC2;
      A     #OutWarning;
      L     8;	//Code=StWarning 
      JC    STC9;
      L     3;	//Code: StStarted
      JU    STC9;
//--------------------
STC2: AN    #StStarting;
      JC    STC3;
      L     2;	// Code: StStarting
      JU    STC9;
//--------------------
STC3: AN    #StFalse;
      JC    STC8;
      L     5;	// Code: StFalse
      JU    STC9;
//--------------------
STC8: L     32;	// Code: StFault
STC9: L     #StCode;	// Old state code
      TAK;
      T     #StCode;	// Save state code
      <>I;
      L     3;	// Load code for CBit methode
      CC    "SYS_CBitCtrl";
END_FUNCTION_BLOCK

